LIN {X 0,Y 291.318,Z 1128.416,A -85,B 0,C 180,E1 14289.507,E2 14289.507} C_VEL
LIN {X 0,Y 294.597,Z 1120.605,A -85,B 0,C 180,E1 14284.989,E2 14284.989} C_VEL
LIN {X 0,Y 299.216,Z 1110.98,A -85,B 0,C 180,E1 14280.578,E2 14280.578} C_VEL
LIN {X 0,Y 304.532,Z 1100.924,A -85,B 0,C 180,E1 14276.748,E2 14276.748} C_VEL
LIN {X 0,Y 312.055,Z 1087.317,A -85,B 0,C 180,E1 14272.497,E2 14272.497} C_VEL
LIN {X 0,Y 318.965,Z 1075.015,A -85,B 0,C 180,E1 14269.304,E2 14269.304} C_VEL
LIN {X 0,Y 328.289,Z 1058.31,A -85,B 0,C 180,E1 14265.705,E2 14265.705} C_VEL
LIN {X 0,Y 336.427,Z 1043.264,A -85,B 0,C 180,E1 14263.018,E2 14263.018} C_VEL
LIN {X 0,Y 345.957,Z 1024.879,A -85,B 0,C 180,E1 14260.269,E2 14260.269} C_VEL
LIN {X 0,Y 354.466,Z 1007.296,A -85,B 0,C 180,E1 14258.092,E2 14258.092} C_VEL
LIN {X 0,Y 363.463,Z 987.421,A -85,B 0,C 180,E1 14256.021,E2 14256.021} C_VEL
LIN {X 0,Y 371.644,Z 967.379,A -85,B 0,C 180,E1 14254.313,E2 14254.313} C_VEL
LIN {X 0,Y 379.169,Z 947.195,A -85,B 0,C 180,E1 14252.87,E2 14252.87} C_VEL
LIN {X 0,Y 386.589,Z 924.342,A -85,B 0,C 180,E1 14251.544,E2 14251.544} C_VEL
LIN {X 0,Y 392.137,Z 904.806,A -85,B 0,C 180,E1 14250.618,E2 14250.618} C_VEL
LIN {X 0,Y 398.28,Z 879.112,A -85,B 0,C 180,E1 14249.658,E2 14249.658} C_VEL
LIN {X 0,Y 402.39,Z 857.399,A -85,B 0,C 180,E1 14249.039,E2 14249.039} C_VEL
LIN {X 0,Y 405.943,Z 831.436,A -85,B 0,C 180,E1 14248.465,E2 14248.465} C_VEL
LIN {X 0,Y 413.005,Z 740.206,A -85,B 0,C 180,E1 14246.94,E2 14246.94} C_VEL
LIN {X 0,Y 422.684,Z 613.309,A -85,B 0,C 180,E1 14244.865,E2 14244.865} C_VEL
LIN {X 0,Y 415.721,Z 599.338,A -85,B 0,C 180,E1 14242.298,E2 14242.298} C_VEL
LIN {X 0,Y 409.613,Z 587.739,A -85,B 0,C 180,E1 14239.76,E2 14239.76} C_VEL
LIN {X 0,Y 404.109,Z 578.023,A -85,B 0,C 180,E1 14237.161,E2 14237.161} C_VEL
LIN {X 0,Y 399.634,Z 571.534,A -85,B 0,C 180,E1 14234.786,E2 14234.786} C_VEL
LIN {X 0,Y 396.985,Z 567.648,A -85,B 0,C 180,E1 14233.176,E2 14233.176} C_VEL
LIN {X 0,Y 393.841,Z 563.029,A -85,B 0,C 180,E1 14230.977,E2 14230.977} C_VEL
LIN {X 0,Y 390.748,Z 558.424,A -85,B 0,C 180,E1 14228.313,E2 14228.313} C_VEL
LIN {X 0,Y 387.61,Z 554.339,A -85,B 0,C 180,E1 14224.587,E2 14224.587} C_VEL
LIN {X 0,Y 387.003,Z 552.755,A -85,B 0,C 180,E1 14223.407,E2 14223.407} C_VEL
LIN {X 0,Y 385.579,Z 551.937,A -85,B 0,C 180,E1 14217.325,E2 14217.325} C_VEL
LIN {X 0,Y 387.13,Z 552.997,A -85,B 0,C 180,E1 14212.804,E2 14212.804} C_VEL
LIN {X 0,Y 389.137,Z 556.879,A -85,B 0,C 180,E1 14209.778,E2 14209.778} C_VEL
LIN {X 0,Y 390.847,Z 558.677,A -85,B 0,C 180,E1 14208.04,E2 14208.04} C_VEL
LIN {X 0,Y 393.889,Z 563.127,A -85,B 0,C 180,E1 14205.445,E2 14205.445} C_VEL
LIN {X 0,Y 398.297,Z 569.544,A -85,B 0,C 180,E1 14202.467,E2 14202.467} C_VEL
LIN {X 0,Y 402.044,Z 575.153,A -85,B 0,C 180,E1 14200.344,E2 14200.344} C_VEL
LIN {X 0,Y 406.988,Z 582.534,A -85,B 0,C 180,E1 14197.92,E2 14197.92} C_VEL
LIN {X 0,Y 414.502,Z 594.463,A -85,B 0,C 180,E1 14194.752,E2 14194.752} C_VEL
LIN {X 0,Y 422.345,Z 607.879,A -85,B 0,C 180,E1 14191.892,E2 14191.892} C_VEL
LIN {X 0,Y 422.901,Z 609.086,A -85,B 0,C 180,E1 14191.695,E2 14191.695} C_VEL
LIN {X 0,Y 406.891,Z 815.861,A -85,B 0,C 180,E1 14188.311,E2 14188.311} C_VEL
LIN {X 0,Y 403.396,Z 842.508,A -85,B 0,C 180,E1 14187.705,E2 14187.705} C_VEL
LIN {X 0,Y 399.622,Z 863.558,A -85,B 0,C 180,E1 14187.058,E2 14187.058} C_VEL
LIN {X 0,Y 394.223,Z 887.589,A -85,B 0,C 180,E1 14186.117,E2 14186.117} C_VEL
LIN {X 0,Y 388.753,Z 907.638,A -85,B 0,C 180,E1 14185.134,E2 14185.134} C_VEL
LIN {X 0,Y 382.006,Z 929.3,A -85,B 0,C 180,E1 14183.852,E2 14183.852} C_VEL
LIN {X 0,Y 374.455,Z 950.085,A -85,B 0,C 180,E1 14182.348,E2 14182.348} C_VEL
LIN {X 0,Y 366.884,Z 968.981,A -85,B 0,C 180,E1 14180.715,E2 14180.715} C_VEL
LIN {X 0,Y 357.58,Z 989.896,A -85,B 0,C 180,E1 14178.539,E2 14178.539} C_VEL
LIN {X 0,Y 349.566,Z 1006.457,A -85,B 0,C 180,E1 14176.478,E2 14176.478} C_VEL
LIN {X 0,Y 339.978,Z 1024.981,A -85,B 0,C 180,E1 14173.721,E2 14173.721} C_VEL
LIN {X 0,Y 331.81,Z 1039.815,A -85,B 0,C 180,E1 14171.066,E2 14171.066} C_VEL
LIN {X 0,Y 323.054,Z 1055.197,A -85,B 0,C 180,E1 14167.795,E2 14167.795} C_VEL
LIN {X 0,Y 315.261,Z 1068.407,A -85,B 0,C 180,E1 14164.371,E2 14164.371} C_VEL
LIN {X 0,Y 307.881,Z 1081.062,A -85,B 0,C 180,E1 14160.44,E2 14160.44} C_VEL
LIN {X 0,Y 301.727,Z 1091.661,A -85,B 0,C 180,E1 14156.363,E2 14156.363} C_VEL
LIN {X 0,Y 296.66,Z 1101.087,A -85,B 0,C 180,E1 14151.97,E2 14151.97} C_VEL
LIN {X 0,Y 292.914,Z 1108.615,A -85,B 0,C 180,E1 14147.482,E2 14147.482} C_VEL
LIN {X 0,Y 290.432,Z 1114.59,A -85,B 0,C 180,E1 14143.016,E2 14143.016} C_VEL
LIN {X 0,Y 288.888,Z 1119.317,A -85,B 0,C 180,E1 14138.15,E2 14138.15} C_VEL
LIN {X 0,Y 288.298,Z 1121.988,A -85,B 0,C 180,E1 14134.177,E2 14134.177} C_VEL
LIN {X 0,Y 288.124,Z 1123.632,A -85,B 0,C 180,E1 14130.199,E2 14130.199} C_VEL
LIN {X 0,Y 288.073,Z 1124.223,A -85,B 0,C 180,E1 14125.621,E2 14125.621} C_VEL
LIN {X 0,Y 288.237,Z 1123.469,A -85,B 0,C 180,E1 14121.366,E2 14121.366} C_VEL
LIN {X 0,Y 288.657,Z 1121.74,A -85,B 0,C 180,E1 14117.395,E2 14117.395} C_VEL
LIN {X 0,Y 289.943,Z 1118.252,A -85,B 0,C 180,E1 14112.541,E2 14112.541} C_VEL
LIN {X 0,Y 292.111,Z 1113.467,A -85,B 0,C 180,E1 14108.069,E2 14108.069} C_VEL
LIN {X 0,Y 295.421,Z 1107.398,A -85,B 0,C 180,E1 14103.68,E2 14103.68} C_VEL
LIN {X 0,Y 300.504,Z 1098.901,A -85,B 0,C 180,E1 14098.953,E2 14098.953} C_VEL
LIN {X 0,Y 306.297,Z 1089.902,A -85,B 0,C 180,E1 14094.932,E2 14094.932} C_VEL
LIN {X 0,Y 314.024,Z 1078.102,A -85,B 0,C 180,E1 14090.681,E2 14090.681} C_VEL
LIN {X 0,Y 321.519,Z 1066.718,A -85,B 0,C 180,E1 14087.316,E2 14087.316} C_VEL
LIN {X 0,Y 331.369,Z 1051.399,A -85,B 0,C 180,E1 14083.598,E2 14083.598} C_VEL
LIN {X 0,Y 339.824,Z 1037.756,A -85,B 0,C 180,E1 14080.87,E2 14080.87} C_VEL
LIN {X 0,Y 350.085,Z 1020.363,A -85,B 0,C 180,E1 14077.973,E2 14077.973} C_VEL
LIN {X 0,Y 359.032,Z 1004.061,A -85,B 0,C 180,E1 14075.726,E2 14075.726} C_VEL
LIN {X 0,Y 368.488,Z 985.668,A -85,B 0,C 180,E1 14073.587,E2 14073.587} C_VEL
LIN {X 0,Y 377.392,Z 966.348,A -85,B 0,C 180,E1 14071.735,E2 14071.735} C_VEL
LIN {X 0,Y 385.777,Z 946.452,A -85,B 0,C 180,E1 14070.131,E2 14070.131} C_VEL
LIN {X 0,Y 393.826,Z 924.602,A -85,B 0,C 180,E1 14068.694,E2 14068.694} C_VEL
LIN {X 0,Y 400.441,Z 904.114,A -85,B 0,C 180,E1 14067.572,E2 14067.572} C_VEL
LIN {X 0,Y 407.002,Z 879.98,A -85,B 0,C 180,E1 14066.509,E2 14066.509} C_VEL
LIN {X 0,Y 411.754,Z 858.766,A -85,B 0,C 180,E1 14065.772,E2 14065.772} C_VEL
LIN {X 0,Y 416.215,Z 833.027,A -85,B 0,C 180,E1 14065.084,E2 14065.084} C_VEL
LIN {X 0,Y 417.621,Z 822.757,A -85,B 0,C 180,E1 14064.861,E2 14064.861} C_VEL
LIN {X 0,Y 418.116,Z 815.259,A -85,B 0,C 180,E1 14064.593,E2 14064.593} C_VEL
LIN {X 0,Y 417.112,Z 795.608,A -85,B 0,C 180,E1 14063.491,E2 14063.491} C_VEL
LIN {X 0,Y 417.306,Z 789.105,A -85,B 0,C 180,E1 14063.295,E2 14063.295} C_VEL
LIN {X 0,Y 431.206,Z 621.77,A -85,B 0,C 180,E1 14060.638,E2 14060.638} C_VEL
LIN {X 0,Y 425.225,Z 611.601,A -85,B 0,C 180,E1 14058.047,E2 14058.047} C_VEL
LIN {X 0,Y 420.08,Z 603.181,A -85,B 0,C 180,E1 14055.461,E2 14055.461} C_VEL
LIN {X 0,Y 415.509,Z 595.786,A -85,B 0,C 180,E1 14052.72,E2 14052.72} C_VEL
LIN {X 0,Y 412.212,Z 590.841,A -85,B 0,C 180,E1 14050.341,E2 14050.341} C_VEL
LIN {X 0,Y 409.345,Z 586.345,A -85,B 0,C 180,E1 14047.721,E2 14047.721} C_VEL
LIN {X 0,Y 406.77,Z 582.311,A -85,B 0,C 180,E1 14044.37,E2 14044.37} C_VEL
LIN {X 0,Y 406.343,Z 581.334,A -85,B 0,C 180,E1 14043.527,E2 14043.527} C_VEL
LIN {X 0,Y 405.047,Z 580.42,A -85,B 0,C 180,E1 14038.161,E2 14038.161} C_VEL
LIN {X 0,Y 406.537,Z 581.568,A -85,B 0,C 180,E1 14033.575,E2 14033.575} C_VEL
LIN {X 0,Y 408.82,Z 585.774,A -85,B 0,C 180,E1 14030.284,E2 14030.284} C_VEL
LIN {X 0,Y 409.908,Z 587.173,A -85,B 0,C 180,E1 14029.174,E2 14029.174} C_VEL
LIN {X 0,Y 413.207,Z 592.327,A -85,B 0,C 180,E1 14026.353,E2 14026.353} C_VEL
LIN {X 0,Y 416.68,Z 597.764,A -85,B 0,C 180,E1 14023.981,E2 14023.981} C_VEL
LIN {X 0,Y 421.249,Z 606.254,A -85,B 0,C 180,E1 14021.31,E2 14021.31} C_VEL
LIN {X 0,Y 426.021,Z 615.589,A -85,B 0,C 180,E1 14018.919,E2 14018.919} C_VEL
LIN {X 0,Y 431.055,Z 625.938,A -85,B 0,C 180,E1 14016.694,E2 14016.694} C_VEL
LIN {X 0,Y 414.036,Z 829.301,A -85,B 0,C 180,E1 14013.439,E2 14013.439} C_VEL
LIN {X 0,Y 410.198,Z 856.084,A -85,B 0,C 180,E1 14012.885,E2 14012.885} C_VEL
LIN {X 0,Y 405.917,Z 877.423,A -85,B 0,C 180,E1 14012.32,E2 14012.32} C_VEL
LIN {X 0,Y 399.909,Z 901.403,A -85,B 0,C 180,E1 14011.505,E2 14011.505} C_VEL
LIN {X 0,Y 393.63,Z 922.113,A -85,B 0,C 180,E1 14010.608,E2 14010.608} C_VEL
LIN {X 0,Y 386.08,Z 944.003,A -85,B 0,C 180,E1 14009.444,E2 14009.444} C_VEL
LIN {X 0,Y 377.335,Z 965.835,A -85,B 0,C 180,E1 14007.991,E2 14007.991} C_VEL
LIN {X 0,Y 368.463,Z 985.839,A -85,B 0,C 180,E1 14006.386,E2 14006.386} C_VEL
LIN {X 0,Y 358.485,Z 1006.049,A -85,B 0,C 180,E1 14004.396,E2 14004.396} C_VEL
LIN {X 0,Y 349.213,Z 1023.426,A -85,B 0,C 180,E1 14002.345,E2 14002.345} C_VEL
LIN {X 0,Y 338.447,Z 1042.153,A -85,B 0,C 180,E1 13999.661,E2 13999.661} C_VEL
LIN {X 0,Y 329.258,Z 1057.274,A -85,B 0,C 180,E1 13997.044,E2 13997.044} C_VEL
LIN {X 0,Y 318.775,Z 1073.827,A -85,B 0,C 180,E1 13993.567,E2 13993.567} C_VEL
LIN {X 0,Y 310.538,Z 1086.484,A -85,B 0,C 180,E1 13990.331,E2 13990.331} C_VEL
LIN {X 0,Y 301.758,Z 1099.978,A -85,B 0,C 180,E1 13986.144,E2 13986.144} C_VEL
LIN {X 0,Y 295.089,Z 1110.433,A -85,B 0,C 180,E1 13982.14,E2 13982.14} C_VEL
LIN {X 0,Y 289.07,Z 1120.545,A -85,B 0,C 180,E1 13977.39,E2 13977.39} C_VEL
LIN {X 0,Y 285.018,Z 1128.059,A -85,B 0,C 180,E1 13972.918,E2 13972.918} C_VEL
LIN {X 0,Y 282.106,Z 1134.694,A -85,B 0,C 180,E1 13967.961,E2 13967.961} C_VEL
LIN {X 0,Y 280.589,Z 1139.286,A -85,B 0,C 180,E1 13963.183,E2 13963.183} C_VEL
LIN {X 0,Y 280.078,Z 1142.124,A -85,B 0,C 180,E1 13959.038,E2 13959.038} C_VEL
LIN {X 0,Y 280.013,Z 1144.004,A -85,B 0,C 180,E1 13954.506,E2 13954.506} C_VEL
LIN {X 0,Y 280.074,Z 1144.409,A -85,B 0,C 180,E1 13950.205,E2 13950.205} C_VEL
LIN {X 0,Y 280.045,Z 1143.704,A -85,B 0,C 180,E1 13946.315,E2 13946.315} C_VEL
LIN {X 0,Y 280.021,Z 1142.095,A -85,B 0,C 180,E1 13942.614,E2 13942.614} C_VEL
LIN {X 0,Y 280.283,Z 1139.39,A -85,B 0,C 180,E1 13938.685,E2 13938.685} C_VEL
LIN {X 0,Y 281.319,Z 1134.776,A -85,B 0,C 180,E1 13933.905,E2 13933.905} C_VEL
LIN {X 0,Y 283.489,Z 1128.378,A -85,B 0,C 180,E1 13929.131,E2 13929.131} C_VEL
LIN {X 0,Y 286.643,Z 1121.177,A -85,B 0,C 180,E1 13924.813,E2 13924.813} C_VEL
LIN {X 0,Y 291.754,Z 1111.066,A -85,B 0,C 180,E1 13919.976,E2 13919.976} C_VEL
LIN {X 0,Y 297.297,Z 1101.056,A -85,B 0,C 180,E1 13916.061,E2 13916.061} C_VEL
LIN {X 0,Y 305.115,Z 1087.545,A -85,B 0,C 180,E1 13911.73,E2 13911.73} C_VEL
LIN {X 0,Y 312.276,Z 1075.296,A -85,B 0,C 180,E1 13908.486,E2 13908.486} C_VEL
LIN {X 0,Y 321.302,Z 1059.818,A -85,B 0,C 180,E1 13905.055,E2 13905.055} C_VEL
LIN {X 0,Y 329.779,Z 1044.674,A -85,B 0,C 180,E1 13902.285,E2 13902.285} C_VEL
LIN {X 0,Y 338.983,Z 1027.674,A -85,B 0,C 180,E1 13899.658,E2 13899.658} C_VEL
LIN {X 0,Y 348.447,Z 1008.81,A -85,B 0,C 180,E1 13897.263,E2 13897.263} C_VEL
LIN {X 0,Y 356.802,Z 991.001,A -85,B 0,C 180,E1 13895.364,E2 13895.364} C_VEL
LIN {X 0,Y 366.103,Z 969.234,A -85,B 0,C 180,E1 13893.449,E2 13893.449} C_VEL
LIN {X 0,Y 373.437,Z 950.196,A -85,B 0,C 180,E1 13892.065,E2 13892.065} C_VEL
LIN {X 0,Y 381.343,Z 927.037,A -85,B 0,C 180,E1 13890.68,E2 13890.68} C_VEL
LIN {X 0,Y 387.34,Z 906.608,A -85,B 0,C 180,E1 13889.697,E2 13889.697} C_VEL
LIN {X 0,Y 393.371,Z 882.74,A -85,B 0,C 180,E1 13888.777,E2 13888.777} C_VEL
LIN {X 0,Y 398.041,Z 859.048,A -85,B 0,C 180,E1 13888.091,E2 13888.091} C_VEL
LIN {X 0,Y 401.696,Z 834.331,A -85,B 0,C 180,E1 13887.53,E2 13887.53} C_VEL
LIN {X 0,Y 405.94,Z 782.941,A -85,B 0,C 180,E1 13886.658,E2 13886.658} C_VEL
LIN {X 0,Y 418.812,Z 617.464,A -85,B 0,C 180,E1 13883.945,E2 13883.945} C_VEL
LIN {X 0,Y 412.599,Z 604.766,A -85,B 0,C 180,E1 13881.54,E2 13881.54} C_VEL
LIN {X 0,Y 406.933,Z 593.772,A -85,B 0,C 180,E1 13879.075,E2 13879.075} C_VEL
LIN {X 0,Y 401.952,Z 584.841,A -85,B 0,C 180,E1 13876.623,E2 13876.623} C_VEL
LIN {X 0,Y 396.118,Z 575.974,A -85,B 0,C 180,E1 13873.28,E2 13873.28} C_VEL
LIN {X 0,Y 392.286,Z 570.526,A -85,B 0,C 180,E1 13870.575,E2 13870.575} C_VEL
LIN {X 0,Y 389.241,Z 565.913,A -85,B 0,C 180,E1 13867.825,E2 13867.825} C_VEL
LIN {X 0,Y 386.492,Z 562.133,A -85,B 0,C 180,E1 13864.377,E2 13864.377} C_VEL
LIN {X 0,Y 385.863,Z 560.619,A -85,B 0,C 180,E1 13863.119,E2 13863.119} C_VEL
LIN {X 0,Y 384.612,Z 559.887,A -85,B 0,C 180,E1 13857.238,E2 13857.238} C_VEL
LIN {X 0,Y 386.069,Z 560.932,A -85,B 0,C 180,E1 13852.933,E2 13852.933} C_VEL
LIN {X 0,Y 388.03,Z 564.753,A -85,B 0,C 180,E1 13849.908,E2 13849.908} C_VEL
LIN {X 0,Y 389.641,Z 566.527,A -85,B 0,C 180,E1 13848.228,E2 13848.228} C_VEL
LIN {X 0,Y 393.378,Z 572.138,A -85,B 0,C 180,E1 13845.049,E2 13845.049} C_VEL
LIN {X 0,Y 396.85,Z 577.291,A -85,B 0,C 180,E1 13842.704,E2 13842.704} C_VEL
LIN {X 0,Y 400.86,Z 583.4,A -85,B 0,C 180,E1 13840.397,E2 13840.397} C_VEL
LIN {X 0,Y 406.295,Z 591.861,A -85,B 0,C 180,E1 13837.72,E2 13837.72} C_VEL
LIN {X 0,Y 412.545,Z 602.045,A -85,B 0,C 180,E1 13835.056,E2 13835.056} C_VEL
LIN {X 0,Y 419.042,Z 613.451,A -85,B 0,C 180,E1 13832.606,E2 13832.606} C_VEL
LIN {X 0,Y 402.939,Z 816.204,A -85,B 0,C 180,E1 13829.295,E2 13829.295} C_VEL
LIN {X 0,Y 399.39,Z 842.701,A -85,B 0,C 180,E1 13828.695,E2 13828.695} C_VEL
LIN {X 0,Y 395.555,Z 863.662,A -85,B 0,C 180,E1 13828.055,E2 13828.055} C_VEL
LIN {X 0,Y 389.975,Z 887.969,A -85,B 0,C 180,E1 13827.109,E2 13827.109} C_VEL
LIN {X 0,Y 384.256,Z 908.433,A -85,B 0,C 180,E1 13826.108,E2 13826.108} C_VEL
LIN {X 0,Y 377.03,Z 930.975,A -85,B 0,C 180,E1 13824.768,E2 13824.768} C_VEL
LIN {X 0,Y 369.105,Z 952.049,A -85,B 0,C 180,E1 13823.224,E2 13823.224} C_VEL
LIN {X 0,Y 360.657,Z 972.488,A -85,B 0,C 180,E1 13821.428,E2 13821.428} C_VEL
LIN {X 0,Y 351.729,Z 991.656,A -85,B 0,C 180,E1 13819.379,E2 13819.379} C_VEL
LIN {X 0,Y 342.976,Z 1009.179,A -85,B 0,C 180,E1 13817.156,E2 13817.156} C_VEL
LIN {X 0,Y 333.519,Z 1026.666,A -85,B 0,C 180,E1 13814.477,E2 13814.477} C_VEL
LIN {X 0,Y 325.281,Z 1041.127,A -85,B 0,C 180,E1 13811.839,E2 13811.839} C_VEL
LIN {X 0,Y 315.828,Z 1057.018,A -85,B 0,C 180,E1 13808.355,E2 13808.355} C_VEL
LIN {X 0,Y 308.222,Z 1069.464,A -85,B 0,C 180,E1 13805.044,E2 13805.044} C_VEL
LIN {X 0,Y 300.268,Z 1082.475,A -85,B 0,C 180,E1 13800.852,E2 13800.852} C_VEL
LIN {X 0,Y 294.476,Z 1092.057,A -85,B 0,C 180,E1 13797.065,E2 13797.065} C_VEL
LIN {X 0,Y 289.158,Z 1101.46,A -85,B 0,C 180,E1 13792.571,E2 13792.571} C_VEL
LIN {X 0,Y 285.212,Z 1108.974,A -85,B 0,C 180,E1 13787.969,E2 13787.969} C_VEL
LIN {X 0,Y 282.551,Z 1115.04,A -85,B 0,C 180,E1 13783.298,E2 13783.298} C_VEL
LIN {X 0,Y 280.943,Z 1119.634,A -85,B 0,C 180,E1 13778.391,E2 13778.391} C_VEL
LIN {X 0,Y 280.316,Z 1122.299,A -85,B 0,C 180,E1 13774.296,E2 13774.296} C_VEL
LIN {X 0,Y 280.12,Z 1124,A -85,B 0,C 180,E1 13770,E2 13770} C_VEL
LIN {X 0,Y 280.077,Z 1124.503,A -85,B 0,C 180,E1 13765.495,E2 13765.495} C_VEL
LIN {X 0,Y 280.254,Z 1123.758,A -85,B 0,C 180,E1 13761.175,E2 13761.175} C_VEL
LIN {X 0,Y 280.723,Z 1122.003,A -85,B 0,C 180,E1 13757.033,E2 13757.033} C_VEL
LIN {X 0,Y 282.127,Z 1118.494,A -85,B 0,C 180,E1 13752.041,E2 13752.041} C_VEL
LIN {X 0,Y 284.457,Z 1113.728,A -85,B 0,C 180,E1 13747.471,E2 13747.471} C_VEL
LIN {X 0,Y 288.014,Z 1107.62,A -85,B 0,C 180,E1 13742.949,E2 13742.949} C_VEL
LIN {X 0,Y 293.416,Z 1099.099,A -85,B 0,C 180,E1 13738.116,E2 13738.116} C_VEL
LIN {X 0,Y 299.516,Z 1090.088,A -85,B 0,C 180,E1 13734.016,E2 13734.016} C_VEL
LIN {X 0,Y 307.628,Z 1078.261,A -85,B 0,C 180,E1 13729.698,E2 13729.698} C_VEL
LIN {X 0,Y 315.517,Z 1066.771,A -85,B 0,C 180,E1 13726.265,E2 13726.265} C_VEL
LIN {X 0,Y 325.7,Z 1051.512,A -85,B 0,C 180,E1 13722.541,E2 13722.541} C_VEL
LIN {X 0,Y 334.627,Z 1037.599,A -85,B 0,C 180,E1 13719.751,E2 13719.751} C_VEL
LIN {X 0,Y 345.645,Z 1019.407,A -85,B 0,C 180,E1 13716.744,E2 13716.744} C_VEL
LIN {X 0,Y 354.289,Z 1004.095,A -85,B 0,C 180,E1 13714.645,E2 13714.645} C_VEL
LIN {X 0,Y 364.331,Z 984.981,A -85,B 0,C 180,E1 13712.443,E2 13712.443} C_VEL
LIN {X 0,Y 373.15,Z 966.298,A -85,B 0,C 180,E1 13710.666,E2 13710.666} C_VEL
LIN {X 0,Y 381.967,Z 945.852,A -85,B 0,C 180,E1 13709.034,E2 13709.034} C_VEL
LIN {X 0,Y 389.918,Z 924.616,A -85,B 0,C 180,E1 13707.655,E2 13707.655} C_VEL
LIN {X 0,Y 396.746,Z 903.886,A -85,B 0,C 180,E1 13706.532,E2 13706.532} C_VEL
LIN {X 0,Y 403.264,Z 880.337,A -85,B 0,C 180,E1 13705.506,E2 13705.506} C_VEL
LIN {X 0,Y 408.135,Z 859.024,A -85,B 0,C 180,E1 13704.772,E2 13704.772} C_VEL
LIN {X 0,Y 412.708,Z 833.11,A -85,B 0,C 180,E1 13704.087,E2 13704.087} C_VEL
LIN {X 0,Y 415.407,Z 810.984,A -85,B 0,C 180,E1 13703.654,E2 13703.654} C_VEL
LIN {X 0,Y 417.306,Z 789.105,A -85,B 0,C 180,E1 13703.295,E2 13703.295} C_VEL
LIN {X 0,Y 417.512,Z 781.549,A -85,B 0,C 180,E1 13703.05,E2 13703.05} C_VEL
LIN {X 0,Y 416.613,Z 761.884,A -85,B 0,C 180,E1 13701.951,E2 13701.951} C_VEL
LIN {X 0,Y 416.864,Z 755.387,A -85,B 0,C 180,E1 13701.753,E2 13701.753} C_VEL
LIN {X 0,Y 427.803,Z 626.61,A -85,B 0,C 180,E1 13699.704,E2 13699.704} C_VEL
LIN {X 0,Y 421.397,Z 615.499,A -85,B 0,C 180,E1 13696.721,E2 13696.721} C_VEL
LIN {X 0,Y 416.189,Z 606.964,A -85,B 0,C 180,E1 13693.83,E2 13693.83} C_VEL
LIN {X 0,Y 413.107,Z 602.1,A -85,B 0,C 180,E1 13691.802,E2 13691.802} C_VEL
LIN {X 0,Y 410.882,Z 598.535,A -85,B 0,C 180,E1 13690.091,E2 13690.091} C_VEL
LIN {X 0,Y 408.093,Z 594.095,A -85,B 0,C 180,E1 13687.461,E2 13687.461} C_VEL
LIN {X 0,Y 405.602,Z 589.9,A -85,B 0,C 180,E1 13684.029,E2 13684.029} C_VEL
LIN {X 0,Y 405.215,Z 589.2,A -85,B 0,C 180,E1 13683.254,E2 13683.254} C_VEL
LIN {X 0,Y 404.072,Z 588.361,A -85,B 0,C 180,E1 13678.157,E2 13678.157} C_VEL
LIN {X 0,Y 405.481,Z 589.489,A -85,B 0,C 180,E1 13673.7,E2 13673.7} C_VEL
LIN {X 0,Y 407.849,Z 593.795,A -85,B 0,C 180,E1 13670.261,E2 13670.261} C_VEL
LIN {X 0,Y 408.78,Z 595.147,A -85,B 0,C 180,E1 13669.286,E2 13669.286} C_VEL
LIN {X 0,Y 411.86,Z 600.037,A -85,B 0,C 180,E1 13666.594,E2 13666.594} C_VEL
LIN {X 0,Y 415.156,Z 605.315,A -85,B 0,C 180,E1 13664.279,E2 13664.279} C_VEL
LIN {X 0,Y 419.675,Z 614.012,A -85,B 0,C 180,E1 13661.562,E2 13661.562} C_VEL
LIN {X 0,Y 424.084,Z 622.914,A -85,B 0,C 180,E1 13659.288,E2 13659.288} C_VEL
LIN {X 0,Y 427.699,Z 630.623,A -85,B 0,C 180,E1 13657.612,E2 13657.612} C_VEL
LIN {X 0,Y 410.688,Z 828.978,A -85,B 0,C 180,E1 13654.455,E2 13654.455} C_VEL
LIN {X 0,Y 406.787,Z 855.739,A -85,B 0,C 180,E1 13653.907,E2 13653.907} C_VEL
LIN {X 0,Y 402.42,Z 877.127,A -85,B 0,C 180,E1 13653.348,E2 13653.348} C_VEL
LIN {X 0,Y 396.146,Z 901.625,A -85,B 0,C 180,E1 13652.524,E2 13652.524} C_VEL
LIN {X 0,Y 389.747,Z 922.274,A -85,B 0,C 180,E1 13651.638,E2 13651.638} C_VEL
LIN {X 0,Y 381.681,Z 945.036,A -85,B 0,C 180,E1 13650.429,E2 13650.429} C_VEL
LIN {X 0,Y 372.956,Z 966.221,A -85,B 0,C 180,E1 13649.019,E2 13649.019} C_VEL
LIN {X 0,Y 363.433,Z 987.13,A -85,B 0,C 180,E1 13647.339,E2 13647.339} C_VEL
LIN {X 0,Y 353.473,Z 1006.609,A -85,B 0,C 180,E1 13645.404,E2 13645.404} C_VEL
LIN {X 0,Y 343.352,Z 1025.024,A -85,B 0,C 180,E1 13643.211,E2 13643.211} C_VEL
LIN {X 0,Y 332.609,Z 1042.975,A -85,B 0,C 180,E1 13640.588,E2 13640.588} C_VEL
LIN {X 0,Y 323.162,Z 1057.999,A -85,B 0,C 180,E1 13637.952,E2 13637.952} C_VEL
LIN {X 0,Y 312.409,Z 1074.294,A -85,B 0,C 180,E1 13634.461,E2 13634.461} C_VEL
LIN {X 0,Y 303.842,Z 1086.956,A -85,B 0,C 180,E1 13631.16,E2 13631.16} C_VEL
LIN {X 0,Y 294.734,Z 1100.306,A -85,B 0,C 180,E1 13626.904,E2 13626.904} C_VEL
LIN {X 0,Y 288.105,Z 1110.228,A -85,B 0,C 180,E1 13623.017,E2 13623.017} C_VEL
LIN {X 0,Y 281.748,Z 1120.319,A -85,B 0,C 180,E1 13618.165,E2 13618.165} C_VEL
LIN {X 0,Y 277.43,Z 1127.824,A -85,B 0,C 180,E1 13613.582,E2 13613.582} C_VEL
LIN {X 0,Y 274.313,Z 1134.442,A -85,B 0,C 180,E1 13608.489,E2 13608.489} C_VEL
LIN {X 0,Y 272.666,Z 1139.027,A -85,B 0,C 180,E1 13603.574,E2 13603.574} C_VEL
LIN {X 0,Y 272.091,Z 1141.858,A -85,B 0,C 180,E1 13599.305,E2 13599.305} C_VEL
LIN {X 0,Y 272.012,Z 1143.731,A -85,B 0,C 180,E1 13594.639,E2 13594.639} C_VEL
LIN {X 0,Y 272.079,Z 1144.12,A -85,B 0,C 180,E1 13590.211,E2 13590.211} C_VEL
LIN {X 0,Y 272.049,Z 1143.407,A -85,B 0,C 180,E1 13586.207,E2 13586.207} C_VEL
LIN {X 0,Y 272.025,Z 1141.787,A -85,B 0,C 180,E1 13582.396,E2 13582.396} C_VEL
LIN {X 0,Y 272.322,Z 1139.071,A -85,B 0,C 180,E1 13578.349,E2 13578.349} C_VEL
LIN {X 0,Y 273.507,Z 1134.284,A -85,B 0,C 180,E1 13573.301,E2 13573.301} C_VEL
LIN {X 0,Y 275.802,Z 1128.026,A -85,B 0,C 180,E1 13568.521,E2 13568.521} C_VEL
LIN {X 0,Y 279.356,Z 1120.449,A -85,B 0,C 180,E1 13563.88,E2 13563.88} C_VEL
LIN {X 0,Y 284.586,Z 1110.681,A -85,B 0,C 180,E1 13559.138,E2 13559.138} C_VEL
LIN {X 0,Y 290.43,Z 1100.658,A -85,B 0,C 180,E1 13555.145,E2 13555.145} C_VEL
LIN {X 0,Y 298.621,Z 1087.123,A -85,B 0,C 180,E1 13550.74,E2 13550.74} C_VEL
LIN {X 0,Y 306.096,Z 1074.862,A -85,B 0,C 180,E1 13547.454,E2 13547.454} C_VEL
LIN {X 0,Y 315.677,Z 1059.008,A -85,B 0,C 180,E1 13543.922,E2 13543.922} C_VEL
LIN {X 0,Y 324.261,Z 1044.194,A -85,B 0,C 180,E1 13541.201,E2 13541.201} C_VEL
LIN {X 0,Y 333.927,Z 1026.89,A -85,B 0,C 180,E1 13538.523,E2 13538.523} C_VEL
LIN {X 0,Y 343.609,Z 1008.08,A -85,B 0,C 180,E1 13536.146,E2 13536.146} C_VEL
LIN {X 0,Y 352.747,Z 989.085,A -85,B 0,C 180,E1 13534.137,E2 13534.137} C_VEL
LIN {X 0,Y 361.984,Z 967.796,A -85,B 0,C 180,E1 13532.301,E2 13532.301} C_VEL
LIN {X 0,Y 369.508,Z 948.636,A -85,B 0,C 180,E1 13530.929,E2 13530.929} C_VEL
LIN {X 0,Y 377.607,Z 925.152,A -85,B 0,C 180,E1 13529.557,E2 13529.557} C_VEL
LIN {X 0,Y 383.385,Z 905.806,A -85,B 0,C 180,E1 13528.644,E2 13528.644} C_VEL
LIN {X 0,Y 389.481,Z 882.018,A -85,B 0,C 180,E1 13527.741,E2 13527.741} C_VEL
LIN {X 0,Y 394.176,Z 858.584,A -85,B 0,C 180,E1 13527.07,E2 13527.07} C_VEL
LIN {X 0,Y 397.887,Z 833.863,A -85,B 0,C 180,E1 13526.514,E2 13526.514} C_VEL
LIN {X 0,Y 402.316,Z 781.445,A -85,B 0,C 180,E1 13525.628,E2 13525.628} C_VEL
LIN {X 0,Y 415.089,Z 621.78,A -85,B 0,C 180,E1 13523.027,E2 13523.027} C_VEL
LIN {X 0,Y 409.386,Z 609.849,A -85,B 0,C 180,E1 13520.699,E2 13520.699} C_VEL
LIN {X 0,Y 404.231,Z 599.763,A -85,B 0,C 180,E1 13518.346,E2 13518.346} C_VEL
LIN {X 0,Y 400.018,Z 592.019,A -85,B 0,C 180,E1 13516.183,E2 13516.183} C_VEL
LIN {X 0,Y 394.574,Z 583.529,A -85,B 0,C 180,E1 13512.96,E2 13512.96} C_VEL
LIN {X 0,Y 390.844,Z 578.114,A -85,B 0,C 180,E1 13510.242,E2 13510.242} C_VEL
LIN {X 0,Y 387.969,Z 573.664,A -85,B 0,C 180,E1 13507.553,E2 13507.553} C_VEL
LIN {X 0,Y 385.303,Z 569.721,A -85,B 0,C 180,E1 13504.018,E2 13504.018} C_VEL
LIN {X 0,Y 384.809,Z 568.525,A -85,B 0,C 180,E1 13502.979,E2 13502.979} C_VEL
LIN {X 0,Y 383.645,Z 567.837,A -85,B 0,C 180,E1 13497.162,E2 13497.162} C_VEL
LIN {X 0,Y 385.011,Z 568.863,A -85,B 0,C 180,E1 13493.064,E2 13493.064} C_VEL
LIN {X 0,Y 387.059,Z 572.778,A -85,B 0,C 180,E1 13489.883,E2 13489.883} C_VEL
LIN {X 0,Y 388.44,Z 574.374,A -85,B 0,C 180,E1 13488.417,E2 13488.417} C_VEL
LIN {X 0,Y 392.011,Z 579.857,A -85,B 0,C 180,E1 13485.298,E2 13485.298} C_VEL
LIN {X 0,Y 395.411,Z 585.033,A -85,B 0,C 180,E1 13482.942,E2 13482.942} C_VEL
LIN {X 0,Y 400.208,Z 592.352,A -85,B 0,C 180,E1 13480.174,E2 13480.174} C_VEL
LIN {X 0,Y 406.317,Z 602.391,A -85,B 0,C 180,E1 13477.195,E2 13477.195} C_VEL
LIN {X 0,Y 412.267,Z 612.537,A -85,B 0,C 180,E1 13474.693,E2 13474.693} C_VEL
LIN {X 0,Y 415.262,Z 618.162,A -85,B 0,C 180,E1 13473.528,E2 13473.528} C_VEL
LIN {X 0,Y 399.107,Z 816.538,A -85,B 0,C 180,E1 13470.297,E2 13470.297} C_VEL
LIN {X 0,Y 395.484,Z 843.014,A -85,B 0,C 180,E1 13469.702,E2 13469.702} C_VEL
LIN {X 0,Y 391.589,Z 863.864,A -85,B 0,C 180,E1 13469.07,E2 13469.07} C_VEL
LIN {X 0,Y 386.063,Z 887.562,A -85,B 0,C 180,E1 13468.159,E2 13468.159} C_VEL
LIN {X 0,Y 380.21,Z 908.113,A -85,B 0,C 180,E1 13467.165,E2 13467.165} C_VEL
LIN {X 0,Y 373.146,Z 929.789,A -85,B 0,C 180,E1 13465.895,E2 13465.895} C_VEL
LIN {X 0,Y 364.901,Z 951.391,A -85,B 0,C 180,E1 13464.337,E2 13464.337} C_VEL
LIN {X 0,Y 356.951,Z 970.219,A -85,B 0,C 180,E1 13462.707,E2 13462.707} C_VEL
LIN {X 0,Y 347.576,Z 990.162,A -85,B 0,C 180,E1 13460.628,E2 13460.628} C_VEL
LIN {X 0,Y 338.958,Z 1006.994,A -85,B 0,C 180,E1 13458.528,E2 13458.528} C_VEL
LIN {X 0,Y 328.493,Z 1025.983,A -85,B 0,C 180,E1 13455.669,E2 13455.669} C_VEL
LIN {X 0,Y 319.786,Z 1040.782,A -85,B 0,C 180,E1 13452.971,E2 13452.971} C_VEL
LIN {X 0,Y 310.411,Z 1056.098,A -85,B 0,C 180,E1 13449.628,E2 13449.628} C_VEL
LIN {X 0,Y 302.402,Z 1068.659,A -85,B 0,C 180,E1 13446.289,E2 13446.289} C_VEL
LIN {X 0,Y 294.674,Z 1080.842,A -85,B 0,C 180,E1 13442.421,E2 13442.421} C_VEL
LIN {X 0,Y 287.829,Z 1091.56,A -85,B 0,C 180,E1 13438.194,E2 13438.194} C_VEL
LIN {X 0,Y 282.561,Z 1100.291,A -85,B 0,C 180,E1 13434.013,E2 13434.013} C_VEL
LIN {X 0,Y 277.84,Z 1108.744,A -85,B 0,C 180,E1 13428.899,E2 13428.899} C_VEL
LIN {X 0,Y 275.12,Z 1114.399,A -85,B 0,C 180,E1 13424.523,E2 13424.523} C_VEL
LIN {X 0,Y 273.155,Z 1119.495,A -85,B 0,C 180,E1 13419.269,E2 13419.269} C_VEL
LIN {X 0,Y 272.383,Z 1122.39,A -85,B 0,C 180,E1 13414.843,E2 13414.843} C_VEL
LIN {X 0,Y 272.127,Z 1124.034,A -85,B 0,C 180,E1 13410.842,E2 13410.842} C_VEL
LIN {X 0,Y 272.075,Z 1124.772,A -85,B 0,C 180,E1 13406.629,E2 13406.629} C_VEL
LIN {X 0,Y 272.2,Z 1124.353,A -85,B 0,C 180,E1 13401.976,E2 13401.976} C_VEL
LIN {X 0,Y 272.654,Z 1122.7,A -85,B 0,C 180,E1 13397.504,E2 13397.504} C_VEL
LIN {X 0,Y 273.717,Z 1120.009,A -85,B 0,C 180,E1 13393.155,E2 13393.155} C_VEL
LIN {X 0,Y 276.175,Z 1115.2,A -85,B 0,C 180,E1 13387.881,E2 13387.881} C_VEL
LIN {X 0,Y 279.666,Z 1109.324,A -85,B 0,C 180,E1 13383.225,E2 13383.225} C_VEL
LIN {X 0,Y 284.801,Z 1101.69,A -85,B 0,C 180,E1 13378.458,E2 13378.458} C_VEL
LIN {X 0,Y 291.175,Z 1092.539,A -85,B 0,C 180,E1 13374.04,E2 13374.04} C_VEL
LIN {X 0,Y 298.579,Z 1082.3,A -85,B 0,C 180,E1 13369.986,E2 13369.986} C_VEL
LIN {X 0,Y 307.251,Z 1070.158,A -85,B 0,C 180,E1 13366.118,E2 13366.118} C_VEL
LIN {X 0,Y 315.854,Z 1057.916,A -85,B 0,C 180,E1 13362.892,E2 13362.892} C_VEL
LIN {X 0,Y 326.484,Z 1042.158,A -85,B 0,C 180,E1 13359.486,E2 13359.486} C_VEL
LIN {X 0,Y 335.456,Z 1028.118,A -85,B 0,C 180,E1 13356.981,E2 13356.981} C_VEL
LIN {X 0,Y 346.242,Z 1010.231,A -85,B 0,C 180,E1 13354.318,E2 13354.318} C_VEL
LIN {X 0,Y 356.05,Z 992.417,A -85,B 0,C 180,E1 13352.145,E2 13352.145} C_VEL
LIN {X 0,Y 365.991,Z 972.877,A -85,B 0,C 180,E1 13350.153,E2 13350.153} C_VEL
LIN {X 0,Y 374.897,Z 953.096,A -85,B 0,C 180,E1 13348.5,E2 13348.5} C_VEL
LIN {X 0,Y 383.402,Z 932.221,A -85,B 0,C 180,E1 13347.049,E2 13347.049} C_VEL
LIN {X 0,Y 390.986,Z 910.474,A -85,B 0,C 180,E1 13345.816,E2 13345.816} C_VEL
LIN {X 0,Y 396.881,Z 891.067,A -85,B 0,C 180,E1 13344.909,E2 13344.909} C_VEL
LIN {X 0,Y 403.105,Z 866.485,A -85,B 0,C 180,E1 13343.984,E2 13343.984} C_VEL
LIN {X 0,Y 407.318,Z 845.379,A -85,B 0,C 180,E1 13343.366,E2 13343.366} C_VEL
LIN {X 0,Y 411.06,Z 820.861,A -85,B 0,C 180,E1 13342.816,E2 13342.816} C_VEL
LIN {X 0,Y 415.87,Z 767.134,A -85,B 0,C 180,E1 13341.938,E2 13341.938} C_VEL
LIN {X 0,Y 416.864,Z 755.387,A -85,B 0,C 180,E1 13341.753,E2 13341.753} C_VEL
LIN {X 0,Y 417.112,Z 747.832,A -85,B 0,C 180,E1 13341.507,E2 13341.507} C_VEL
LIN {X 0,Y 416.409,Z 728.183,A -85,B 0,C 180,E1 13340.397,E2 13340.397} C_VEL
LIN {X 0,Y 416.7,Z 721.685,A -85,B 0,C 180,E1 13340.201,E2 13340.201} C_VEL
LIN {X 0,Y 424.554,Z 631.643,A -85,B 0,C 180,E1 13338.777,E2 13338.777} C_VEL
LIN {X 0,Y 418.914,Z 621.735,A -85,B 0,C 180,E1 13336.003,E2 13336.003} C_VEL
LIN {X 0,Y 414.212,Z 613.848,A -85,B 0,C 180,E1 13333.257,E2 13333.257} C_VEL
LIN {X 0,Y 411.453,Z 609.352,A -85,B 0,C 180,E1 13331.352,E2 13331.352} C_VEL
LIN {X 0,Y 409.476,Z 606.124,A -85,B 0,C 180,E1 13329.771,E2 13329.771} C_VEL
LIN {X 0,Y 406.982,Z 601.97,A -85,B 0,C 180,E1 13327.34,E2 13327.34} C_VEL
LIN {X 0,Y 404.51,Z 597.696,A -85,B 0,C 180,E1 13323.827,E2 13323.827} C_VEL
LIN {X 0,Y 404.097,Z 597.066,A -85,B 0,C 180,E1 13322.979,E2 13322.979} C_VEL
LIN {X 0,Y 403.106,Z 596.316,A -85,B 0,C 180,E1 13318.01,E2 13318.01} C_VEL
LIN {X 0,Y 404.427,Z 597.407,A -85,B 0,C 180,E1 13313.826,E2 13313.826} C_VEL
LIN {X 0,Y 406.747,Z 601.677,A -85,B 0,C 180,E1 13310.377,E2 13310.377} C_VEL
LIN {X 0,Y 407.654,Z 603.114,A -85,B 0,C 180,E1 13309.4,E2 13309.4} C_VEL
LIN {X 0,Y 410.52,Z 607.744,A -85,B 0,C 180,E1 13306.836,E2 13306.836} C_VEL
LIN {X 0,Y 413.643,Z 612.866,A -85,B 0,C 180,E1 13304.579,E2 13304.579} C_VEL
LIN {X 0,Y 418.347,Z 622.233,A -85,B 0,C 180,E1 13301.681,E2 13301.681} C_VEL
LIN {X 0,Y 423.857,Z 633.728,A -85,B 0,C 180,E1 13298.843,E2 13298.843} C_VEL
LIN {X 0,Y 424.445,Z 635.363,A -85,B 0,C 180,E1 13298.547,E2 13298.547} C_VEL
LIN {X 0,Y 407.454,Z 828.843,A -85,B 0,C 180,E1 13295.484,E2 13295.484} C_VEL
LIN {X 0,Y 403.488,Z 855.505,A -85,B 0,C 180,E1 13294.943,E2 13294.943} C_VEL
LIN {X 0,Y 399.043,Z 876.886,A -85,B 0,C 180,E1 13294.393,E2 13294.393} C_VEL
LIN {X 0,Y 392.511,Z 901.848,A -85,B 0,C 180,E1 13293.563,E2 13293.563} C_VEL
LIN {X 0,Y 385.993,Z 922.435,A -85,B 0,C 180,E1 13292.689,E2 13292.689} C_VEL
LIN {X 0,Y 377.765,Z 945.105,A -85,B 0,C 180,E1 13291.493,E2 13291.493} C_VEL
LIN {X 0,Y 369.012,Z 965.904,A -85,B 0,C 180,E1 13290.122,E2 13290.122} C_VEL
LIN {X 0,Y 359.463,Z 986.41,A -85,B 0,C 180,E1 13288.492,E2 13288.492} C_VEL
LIN {X 0,Y 349.141,Z 1006.138,A -85,B 0,C 180,E1 13286.552,E2 13286.552} C_VEL
LIN {X 0,Y 339.149,Z 1023.841,A -85,B 0,C 180,E1 13284.461,E2 13284.461} C_VEL
LIN {X 0,Y 328.05,Z 1041.936,A -85,B 0,C 180,E1 13281.849,E2 13281.849} C_VEL
LIN {X 0,Y 318.252,Z 1057.023,A -85,B 0,C 180,E1 13279.216,E2 13279.216} C_VEL
LIN {X 0,Y 307.141,Z 1073.319,A -85,B 0,C 180,E1 13275.742,E2 13275.742} C_VEL
LIN {X 0,Y 298.103,Z 1086.145,A -85,B 0,C 180,E1 13272.392,E2 13272.392} C_VEL
LIN {X 0,Y 288.526,Z 1099.59,A -85,B 0,C 180,E1 13268.088,E2 13268.088} C_VEL
LIN {X 0,Y 281.506,Z 1109.557,A -85,B 0,C 180,E1 13264.139,E2 13264.139} C_VEL
LIN {X 0,Y 274.963,Z 1119.371,A -85,B 0,C 180,E1 13259.401,E2 13259.401} C_VEL
LIN {X 0,Y 270.056,Z 1127.278,A -85,B 0,C 180,E1 13254.5,E2 13254.5} C_VEL
LIN {X 0,Y 266.754,Z 1133.699,A -85,B 0,C 180,E1 13249.488,E2 13249.488} C_VEL
LIN {X 0,Y 264.805,Z 1138.6,A -85,B 0,C 180,E1 13244.208,E2 13244.208} C_VEL
LIN {X 0,Y 264.126,Z 1141.472,A -85,B 0,C 180,E1 13239.808,E2 13239.808} C_VEL
LIN {X 0,Y 264.003,Z 1143.314,A -85,B 0,C 180,E1 13235.215,E2 13235.215} C_VEL
LIN {X 0,Y 264.074,Z 1143.875,A -85,B 0,C 180,E1 13230.651,E2 13230.651} C_VEL
LIN {X 0,Y 264.054,Z 1143.178,A -85,B 0,C 180,E1 13226.309,E2 13226.309} C_VEL
LIN {X 0,Y 264.028,Z 1141.596,A -85,B 0,C 180,E1 13222.383,E2 13222.383} C_VEL
LIN {X 0,Y 264.336,Z 1138.917,A -85,B 0,C 180,E1 13218.214,E2 13218.214} C_VEL
LIN {X 0,Y 265.54,Z 1134.338,A -85,B 0,C 180,E1 13213.145,E2 13213.145} C_VEL
LIN {X 0,Y 268.004,Z 1127.987,A -85,B 0,C 180,E1 13208.094,E2 13208.094} C_VEL
LIN {X 0,Y 271.616,Z 1120.663,A -85,B 0,C 180,E1 13203.451,E2 13203.451} C_VEL
LIN {X 0,Y 277.206,Z 1110.766,A -85,B 0,C 180,E1 13198.465,E2 13198.465} C_VEL
LIN {X 0,Y 283.302,Z 1100.789,A -85,B 0,C 180,E1 13194.384,E2 13194.384} C_VEL
LIN {X 0,Y 291.816,Z 1087.351,A -85,B 0,C 180,E1 13189.896,E2 13189.896} C_VEL
LIN {X 0,Y 299.563,Z 1075.143,A -85,B 0,C 180,E1 13186.56,E2 13186.56} C_VEL
LIN {X 0,Y 309.257,Z 1059.753,A -85,B 0,C 180,E1 13183.054,E2 13183.054} C_VEL
LIN {X 0,Y 318.86,Z 1043.714,A -85,B 0,C 180,E1 13180.08,E2 13180.08} C_VEL
LIN {X 0,Y 328.97,Z 1026.151,A -85,B 0,C 180,E1 13177.361,E2 13177.361} C_VEL
LIN {X 0,Y 338.83,Z 1007.503,A -85,B 0,C 180,E1 13175.015,E2 13175.015} C_VEL
LIN {X 0,Y 348.198,Z 988.526,A -85,B 0,C 180,E1 13173.016,E2 13173.016} C_VEL
LIN {X 0,Y 357.205,Z 968.298,A -85,B 0,C 180,E1 13171.278,E2 13171.278} C_VEL
LIN {X 0,Y 364.984,Z 948.986,A -85,B 0,C 180,E1 13169.896,E2 13169.896} C_VEL
LIN {X 0,Y 373.292,Z 925.553,A -85,B 0,C 180,E1 13168.529,E2 13168.529} C_VEL
LIN {X 0,Y 379.185,Z 906.301,A -85,B 0,C 180,E1 13167.623,E2 13167.623} C_VEL
LIN {X 0,Y 385.397,Z 882.768,A -85,B 0,C 180,E1 13166.729,E2 13166.729} C_VEL
LIN {X 0,Y 390.331,Z 858.723,A -85,B 0,C 180,E1 13166.044,E2 13166.044} C_VEL
LIN {X 0,Y 394.118,Z 834.2,A -85,B 0,C 180,E1 13165.494,E2 13165.494} C_VEL
LIN {X 0,Y 398.31,Z 786.317,A -85,B 0,C 180,E1 13164.684,E2 13164.684} C_VEL
LIN {X 0,Y 411.428,Z 626,A -85,B 0,C 180,E1 13162.075,E2 13162.075} C_VEL
LIN {X 0,Y 405.976,Z 614.451,A -85,B 0,C 180,E1 13159.72,E2 13159.72} C_VEL
LIN {X 0,Y 400.48,Z 603.441,A -85,B 0,C 180,E1 13157.022,E2 13157.022} C_VEL
LIN {X 0,Y 397.6,Z 598.453,A -85,B 0,C 180,E1 13155.46,E2 13155.46} C_VEL
LIN {X 0,Y 392.933,Z 590.954,A -85,B 0,C 180,E1 13152.566,E2 13152.566} C_VEL
LIN {X 0,Y 389.503,Z 585.803,A -85,B 0,C 180,E1 13149.979,E2 13149.979} C_VEL
LIN {X 0,Y 386.707,Z 581.415,A -85,B 0,C 180,E1 13147.279,E2 13147.279} C_VEL
LIN {X 0,Y 384.165,Z 577.411,A -85,B 0,C 180,E1 13143.731,E2 13143.731} C_VEL
LIN {X 0,Y 383.758,Z 576.432,A -85,B 0,C 180,E1 13142.838,E2 13142.838} C_VEL
LIN {X 0,Y 382.67,Z 575.779,A -85,B 0,C 180,E1 13137.154,E2 13137.154} C_VEL
LIN {X 0,Y 383.955,Z 576.791,A -85,B 0,C 180,E1 13133.195,E2 13133.195} C_VEL
LIN {X 0,Y 386.088,Z 580.8,A -85,B 0,C 180,E1 13129.857,E2 13129.857} C_VEL
LIN {X 0,Y 387.243,Z 582.218,A -85,B 0,C 180,E1 13128.607,E2 13128.607} C_VEL
LIN {X 0,Y 390.651,Z 587.572,A -85,B 0,C 180,E1 13125.549,E2 13125.549} C_VEL
LIN {X 0,Y 393.872,Z 592.591,A -85,B 0,C 180,E1 13123.254,E2 13123.254} C_VEL
LIN {X 0,Y 398.498,Z 599.852,A -85,B 0,C 180,E1 13120.505,E2 13120.505} C_VEL
LIN {X 0,Y 404.338,Z 609.671,A -85,B 0,C 180,E1 13117.577,E2 13117.577} C_VEL
LIN {X 0,Y 410.079,Z 619.723,A -85,B 0,C 180,E1 13115.091,E2 13115.091} C_VEL
LIN {X 0,Y 411.607,Z 622.679,A -85,B 0,C 180,E1 13114.47,E2 13114.47} C_VEL
LIN {X 0,Y 395.416,Z 816.709,A -85,B 0,C 180,E1 13111.322,E2 13111.322} C_VEL
LIN {X 0,Y 391.702,Z 843.327,A -85,B 0,C 180,E1 13110.727,E2 13110.727} C_VEL
LIN {X 0,Y 387.726,Z 864.173,A -85,B 0,C 180,E1 13110.101,E2 13110.101} C_VEL
LIN {X 0,Y 381.926,Z 888.42,A -85,B 0,C 180,E1 13109.173,E2 13109.173} C_VEL
LIN {X 0,Y 375.951,Z 908.903,A -85,B 0,C 180,E1 13108.185,E2 13108.185} C_VEL
LIN {X 0,Y 368.392,Z 931.468,A -85,B 0,C 180,E1 13106.86,E2 13106.86} C_VEL
LIN {X 0,Y 360.297,Z 952.042,A -85,B 0,C 180,E1 13105.371,E2 13105.371} C_VEL
LIN {X 0,Y 351.835,Z 971.561,A -85,B 0,C 180,E1 13103.677,E2 13103.677} C_VEL
LIN {X 0,Y 342.092,Z 991.586,A -85,B 0,C 180,E1 13101.567,E2 13101.567} C_VEL
LIN {X 0,Y 333.096,Z 1008.624,A -85,B 0,C 180,E1 13099.417,E2 13099.417} C_VEL
LIN {X 0,Y 322.901,Z 1026.482,A -85,B 0,C 180,E1 13096.694,E2 13096.694} C_VEL
LIN {X 0,Y 313.916,Z 1041.264,A -85,B 0,C 180,E1 13093.978,E2 13093.978} C_VEL
LIN {X 0,Y 303.752,Z 1057.234,A -85,B 0,C 180,E1 13090.428,E2 13090.428} C_VEL
LIN {X 0,Y 295.33,Z 1069.963,A -85,B 0,C 180,E1 13086.963,E2 13086.963} C_VEL
LIN {X 0,Y 286.798,Z 1082.79,A -85,B 0,C 180,E1 13082.71,E2 13082.71} C_VEL
LIN {X 0,Y 280.12,Z 1092.848,A -85,B 0,C 180,E1 13078.576,E2 13078.576} C_VEL
LIN {X 0,Y 274.26,Z 1102.202,A -85,B 0,C 180,E1 13073.871,E2 13073.871} C_VEL
LIN {X 0,Y 269.874,Z 1109.691,A -85,B 0,C 180,E1 13069.029,E2 13069.029} C_VEL
LIN {X 0,Y 266.818,Z 1115.92,A -85,B 0,C 180,E1 13063.928,E2 13063.928} C_VEL
LIN {X 0,Y 265.063,Z 1120.28,A -85,B 0,C 180,E1 13058.897,E2 13058.897} C_VEL
LIN {X 0,Y 264.355,Z 1122.922,A -85,B 0,C 180,E1 13054.556,E2 13054.556} C_VEL
LIN {X 0,Y 264.131,Z 1124.6,A -85,B 0,C 180,E1 13050,E2 13050} C_VEL
LIN {X 0,Y 264.088,Z 1125.063,A -85,B 0,C 180,E1 13045.222,E2 13045.222} C_VEL
LIN {X 0,Y 264.286,Z 1124.365,A -85,B 0,C 180,E1 13040.857,E2 13040.857} C_VEL
LIN {X 0,Y 264.798,Z 1122.745,A -85,B 0,C 180,E1 13036.683,E2 13036.683} C_VEL
LIN {X 0,Y 266.281,Z 1119.544,A -85,B 0,C 180,E1 13031.614,E2 13031.614} C_VEL
LIN {X 0,Y 269.125,Z 1114.442,A -85,B 0,C 180,E1 13026.343,E2 13026.343} C_VEL
LIN {X 0,Y 272.922,Z 1108.658,A -85,B 0,C 180,E1 13021.796,E2 13021.796} C_VEL
LIN {X 0,Y 279.03,Z 1100.066,A -85,B 0,C 180,E1 13016.611,E2 13016.611} C_VEL
LIN {X 0,Y 285.501,Z 1091.368,A -85,B 0,C 180,E1 13012.455,E2 13012.455} C_VEL
LIN {X 0,Y 294.709,Z 1079.149,A -85,B 0,C 180,E1 13007.795,E2 13007.795} C_VEL
LIN {X 0,Y 303.17,Z 1067.784,A -85,B 0,C 180,E1 13004.3,E2 13004.3} C_VEL
LIN {X 0,Y 314.194,Z 1052.504,A -85,B 0,C 180,E1 13000.482,E2 13000.482} C_VEL
LIN {X 0,Y 323.548,Z 1038.886,A -85,B 0,C 180,E1 12997.707,E2 12997.707} C_VEL
LIN {X 0,Y 334.803,Z 1021.545,A -85,B 0,C 180,E1 12994.786,E2 12994.786} C_VEL
LIN {X 0,Y 344.55,Z 1005.273,A -85,B 0,C 180,E1 12992.537,E2 12992.537} C_VEL
LIN {X 0,Y 354.785,Z 986.942,A -85,B 0,C 180,E1 12990.413,E2 12990.413} C_VEL
LIN {X 0,Y 364.374,Z 967.676,A -85,B 0,C 180,E1 12988.583,E2 12988.583} C_VEL
LIN {X 0,Y 372.869,Z 948.944,A -85,B 0,C 180,E1 12987.089,E2 12987.089} C_VEL
LIN {X 0,Y 381.596,Z 927.117,A -85,B 0,C 180,E1 12985.66,E2 12985.66} C_VEL
LIN {X 0,Y 388.63,Z 906.839,A -85,B 0,C 180,E1 12984.562,E2 12984.562} C_VEL
LIN {X 0,Y 395.792,Z 882.541,A -85,B 0,C 180,E1 12983.501,E2 12983.501} C_VEL
LIN {X 0,Y 400.974,Z 860.945,A -85,B 0,C 180,E1 12982.763,E2 12982.763} C_VEL
LIN {X 0,Y 405.571,Z 836.84,A -85,B 0,C 180,E1 12982.12,E2 12982.12} C_VEL
LIN {X 0,Y 408.647,Z 813.312,A -85,B 0,C 180,E1 12981.656,E2 12981.656} C_VEL
LIN {X 0,Y 416.7,Z 721.685,A -85,B 0,C 180,E1 12980.201,E2 12980.201} C_VEL
LIN {X 0,Y 416.999,Z 714.132,A -85,B 0,C 180,E1 12979.957,E2 12979.957} C_VEL
LIN {X 0,Y 416.506,Z 694.493,A -85,B 0,C 180,E1 12978.842,E2 12978.842} C_VEL
LIN {X 0,Y 416.828,Z 687.998,A -85,B 0,C 180,E1 12978.644,E2 12978.644} C_VEL
LIN {X 0,Y 421.387,Z 636.678,A -85,B 0,C 180,E1 12977.824,E2 12977.824} C_VEL
LIN {X 0,Y 415.75,Z 626.529,A -85,B 0,C 180,E1 12974.841,E2 12974.841} C_VEL
LIN {X 0,Y 410.932,Z 618.302,A -85,B 0,C 180,E1 12971.723,E2 12971.723} C_VEL
LIN {X 0,Y 408.165,Z 613.814,A -85,B 0,C 180,E1 12969.518,E2 12969.518} C_VEL
LIN {X 0,Y 405.742,Z 609.715,A -85,B 0,C 180,E1 12967.078,E2 12967.078} C_VEL
LIN {X 0,Y 403.365,Z 605.282,A -85,B 0,C 180,E1 12963.482,E2 12963.482} C_VEL
LIN {X 0,Y 402.101,Z 604.24,A -85,B 0,C 180,E1 12958.718,E2 12958.718} C_VEL
LIN {X 0,Y 403.348,Z 605.214,A -85,B 0,C 180,E1 12954.024,E2 12954.024} C_VEL
LIN {X 0,Y 405.648,Z 609.558,A -85,B 0,C 180,E1 12950.494,E2 12950.494} C_VEL
LIN {X 0,Y 406.728,Z 611.467,A -85,B 0,C 180,E1 12949.303,E2 12949.303} C_VEL
LIN {X 0,Y 409.188,Z 615.451,A -85,B 0,C 180,E1 12947.08,E2 12947.08} C_VEL
LIN {X 0,Y 412.14,Z 620.424,A -85,B 0,C 180,E1 12944.882,E2 12944.882} C_VEL
LIN {X 0,Y 417.202,Z 630.788,A -85,B 0,C 180,E1 12941.702,E2 12941.702} C_VEL
LIN {X 0,Y 421.307,Z 640.084,A -85,B 0,C 180,E1 12939.496,E2 12939.496} C_VEL
LIN {X 0,Y 404.376,Z 828.493,A -85,B 0,C 180,E1 12936.533,E2 12936.533} C_VEL
LIN {X 0,Y 400.33,Z 855.236,A -85,B 0,C 180,E1 12935.997,E2 12935.997} C_VEL
LIN {X 0,Y 395.794,Z 876.683,A -85,B 0,C 180,E1 12935.454,E2 12935.454} C_VEL
LIN {X 0,Y 389.401,Z 900.795,A -85,B 0,C 180,E1 12934.67,E2 12934.67} C_VEL
LIN {X 0,Y 382.592,Z 921.953,A -85,B 0,C 180,E1 12933.789,E2 12933.789} C_VEL
LIN {X 0,Y 374.4,Z 944.187,A -85,B 0,C 180,E1 12932.639,E2 12932.639} C_VEL
LIN {X 0,Y 365.419,Z 965.127,A -85,B 0,C 180,E1 12931.281,E2 12931.281} C_VEL
LIN {X 0,Y 355.909,Z 985.13,A -85,B 0,C 180,E1 12929.716,E2 12929.716} C_VEL
LIN {X 0,Y 345.163,Z 1005.295,A -85,B 0,C 180,E1 12927.767,E2 12927.767} C_VEL
LIN {X 0,Y 335.117,Z 1022.659,A -85,B 0,C 180,E1 12925.74,E2 12925.74} C_VEL
LIN {X 0,Y 323.661,Z 1040.898,A -85,B 0,C 180,E1 12923.143,E2 12923.143} C_VEL
LIN {X 0,Y 313.51,Z 1056.048,A -85,B 0,C 180,E1 12920.518,E2 12920.518} C_VEL
LIN {X 0,Y 301.951,Z 1072.458,A -85,B 0,C 180,E1 12917.04,E2 12917.04} C_VEL
LIN {X 0,Y 292.504,Z 1085.335,A -85,B 0,C 180,E1 12913.671,E2 12913.671} C_VEL
LIN {X 0,Y 282.856,Z 1098.353,A -85,B 0,C 180,E1 12909.516,E2 12909.516} C_VEL
LIN {X 0,Y 275.016,Z 1108.885,A -85,B 0,C 180,E1 12905.316,E2 12905.316} C_VEL
LIN {X 0,Y 268.042,Z 1118.778,A -85,B 0,C 180,E1 12900.486,E2 12900.486} C_VEL
LIN {X 0,Y 262.756,Z 1126.732,A -85,B 0,C 180,E1 12895.468,E2 12895.468} C_VEL
LIN {X 0,Y 259.261,Z 1132.932,A -85,B 0,C 180,E1 12890.546,E2 12890.546} C_VEL
LIN {X 0,Y 256.966,Z 1138.174,A -85,B 0,C 180,E1 12884.881,E2 12884.881} C_VEL
LIN {X 0,Y 256.174,Z 1141.086,A -85,B 0,C 180,E1 12880.343,E2 12880.343} C_VEL
LIN {X 0,Y 256.014,Z 1142.897,A -85,B 0,C 180,E1 12875.828,E2 12875.828} C_VEL
LIN {X 0,Y 256.081,Z 1143.623,A -85,B 0,C 180,E1 12871.119,E2 12871.119} C_VEL
LIN {X 0,Y 256.056,Z 1143.02,A -85,B 0,C 180,E1 12866.642,E2 12866.642} C_VEL
LIN {X 0,Y 256.03,Z 1141.406,A -85,B 0,C 180,E1 12862.37,E2 12862.37} C_VEL
LIN {X 0,Y 256.352,Z 1138.764,A -85,B 0,C 180,E1 12858.069,E2 12858.069} C_VEL
LIN {X 0,Y 257.462,Z 1134.651,A -85,B 0,C 180,E1 12853.298,E2 12853.298} C_VEL
LIN {X 0,Y 260.22,Z 1127.948,A -85,B 0,C 180,E1 12847.641,E2 12847.641} C_VEL
LIN {X 0,Y 263.927,Z 1120.815,A -85,B 0,C 180,E1 12842.959,E2 12842.959} C_VEL
LIN {X 0,Y 270.159,Z 1110.38,A -85,B 0,C 180,E1 12837.543,E2 12837.543} C_VEL
LIN {X 0,Y 276.583,Z 1100.382,A -85,B 0,C 180,E1 12833.376,E2 12833.376} C_VEL
LIN {X 0,Y 285.5,Z 1086.928,A -85,B 0,C 180,E1 12828.82,E2 12828.82} C_VEL
LIN {X 0,Y 293.918,Z 1074.205,A -85,B 0,C 180,E1 12825.317,E2 12825.317} C_VEL
LIN {X 0,Y 304.175,Z 1058.425,A -85,B 0,C 180,E1 12821.737,E2 12821.737} C_VEL
LIN {X 0,Y 313.635,Z 1043.151,A -85,B 0,C 180,E1 12818.907,E2 12818.907} C_VEL
LIN {X 0,Y 323.938,Z 1025.783,A -85,B 0,C 180,E1 12816.218,E2 12816.218} C_VEL
LIN {X 0,Y 334.145,Z 1007.005,A -85,B 0,C 180,E1 12813.861,E2 12813.861} C_VEL
LIN {X 0,Y 344.129,Z 987.284,A -85,B 0,C 180,E1 12811.801,E2 12811.801} C_VEL
LIN {X 0,Y 353.635,Z 966.242,A -85,B 0,C 180,E1 12810.031,E2 12810.031} C_VEL
LIN {X 0,Y 362.506,Z 944.5,A -85,B 0,C 180,E1 12808.52,E2 12808.52} C_VEL
LIN {X 0,Y 370.21,Z 922.52,A -85,B 0,C 180,E1 12807.303,E2 12807.303} C_VEL
LIN {X 0,Y 376.638,Z 901.603,A -85,B 0,C 180,E1 12806.364,E2 12806.364} C_VEL
LIN {X 0,Y 382.913,Z 876.88,A -85,B 0,C 180,E1 12805.497,E2 12805.497} C_VEL
LIN {X 0,Y 387.243,Z 855.459,A -85,B 0,C 180,E1 12804.915,E2 12804.915} C_VEL
LIN {X 0,Y 391.124,Z 828.354,A -85,B 0,C 180,E1 12804.342,E2 12804.342} C_VEL
LIN {X 0,Y 407.915,Z 630.315,A -85,B 0,C 180,E1 12801.121,E2 12801.121} C_VEL
LIN {X 0,Y 401.776,Z 617.145,A -85,B 0,C 180,E1 12798.275,E2 12798.275} C_VEL
LIN {X 0,Y 396.723,Z 607.112,A -85,B 0,C 180,E1 12795.57,E2 12795.57} C_VEL
LIN {X 0,Y 391.522,Z 598.635,A -85,B 0,C 180,E1 12792.313,E2 12792.313} C_VEL
LIN {X 0,Y 388.171,Z 593.492,A -85,B 0,C 180,E1 12789.714,E2 12789.714} C_VEL
LIN {X 0,Y 385.592,Z 589.289,A -85,B 0,C 180,E1 12787.15,E2 12787.15} C_VEL
LIN {X 0,Y 383.068,Z 585.205,A -85,B 0,C 180,E1 12783.517,E2 12783.517} C_VEL
LIN {X 0,Y 382.708,Z 584.339,A -85,B 0,C 180,E1 12782.695,E2 12782.695} C_VEL
LIN {X 0,Y 381.695,Z 583.721,A -85,B 0,C 180,E1 12777.147,E2 12777.147} C_VEL
LIN {X 0,Y 382.902,Z 584.715,A -85,B 0,C 180,E1 12773.327,E2 12773.327} C_VEL
LIN {X 0,Y 384.991,Z 588.683,A -85,B 0,C 180,E1 12769.979,E2 12769.979} C_VEL
LIN {X 0,Y 386.051,Z 590.058,A -85,B 0,C 180,E1 12768.799,E2 12768.799} C_VEL
LIN {X 0,Y 389.299,Z 595.288,A -85,B 0,C 180,E1 12765.801,E2 12765.801} C_VEL
LIN {X 0,Y 392.449,Z 600.328,A -85,B 0,C 180,E1 12763.496,E2 12763.496} C_VEL
LIN {X 0,Y 396.925,Z 607.577,A -85,B 0,C 180,E1 12760.769,E2 12760.769} C_VEL
LIN {X 0,Y 402.594,Z 617.323,A -85,B 0,C 180,E1 12757.859,E2 12757.859} C_VEL
LIN {X 0,Y 408.062,Z 627.188,A -85,B 0,C 180,E1 12755.43,E2 12755.43} C_VEL
LIN {X 0,Y 391.831,Z 817.099,A -85,B 0,C 180,E1 12752.361,E2 12752.361} C_VEL
LIN {X 0,Y 388.066,Z 843.546,A -85,B 0,C 180,E1 12751.775,E2 12751.775} C_VEL
LIN {X 0,Y 384.036,Z 864.268,A -85,B 0,C 180,E1 12751.16,E2 12751.16} C_VEL
LIN {X 0,Y 378.137,Z 888.49,A -85,B 0,C 180,E1 12750.244,E2 12750.244} C_VEL
LIN {X 0,Y 371.813,Z 909.692,A -85,B 0,C 180,E1 12749.228,E2 12749.228} C_VEL
LIN {X 0,Y 364.089,Z 932.156,A -85,B 0,C 180,E1 12747.912,E2 12747.912} C_VEL
LIN {X 0,Y 355.812,Z 952.691,A -85,B 0,C 180,E1 12746.431,E2 12746.431} C_VEL
LIN {X 0,Y 346.822,Z 972.9,A -85,B 0,C 180,E1 12744.676,E2 12744.676} C_VEL
LIN {X 0,Y 337.155,Z 992.148,A -85,B 0,C 180,E1 12742.637,E2 12742.637} C_VEL
LIN {X 0,Y 327.616,Z 1009.709,A -85,B 0,C 180,E1 12740.411,E2 12740.411} C_VEL
LIN {X 0,Y 317.416,Z 1026.98,A -85,B 0,C 180,E1 12737.755,E2 12737.755} C_VEL
LIN {X 0,Y 308.145,Z 1041.745,A -85,B 0,C 180,E1 12735.023,E2 12735.023} C_VEL
LIN {X 0,Y 297.633,Z 1057.682,A -85,B 0,C 180,E1 12731.439,E2 12731.439} C_VEL
LIN {X 0,Y 289.06,Z 1070.151,A -85,B 0,C 180,E1 12728.005,E2 12728.005} C_VEL
LIN {X 0,Y 280.353,Z 1082.714,A -85,B 0,C 180,E1 12723.798,E2 12723.798} C_VEL
LIN {X 0,Y 273.327,Z 1092.796,A -85,B 0,C 180,E1 12719.595,E2 12719.595} C_VEL
LIN {X 0,Y 267.108,Z 1102.226,A -85,B 0,C 180,E1 12714.788,E2 12714.788} C_VEL
LIN {X 0,Y 262.302,Z 1109.942,A -85,B 0,C 180,E1 12709.684,E2 12709.684} C_VEL
LIN {X 0,Y 259.083,Z 1116.078,A -85,B 0,C 180,E1 12704.528,E2 12704.528} C_VEL
LIN {X 0,Y 257.131,Z 1120.603,A -85,B 0,C 180,E1 12699.174,E2 12699.174} C_VEL
LIN {X 0,Y 256.376,Z 1123.233,A -85,B 0,C 180,E1 12694.698,E2 12694.698} C_VEL
LIN {X 0,Y 256.136,Z 1124.901,A -85,B 0,C 180,E1 12690,E2 12690} C_VEL
LIN {X 0,Y 256.095,Z 1125.343,A -85,B 0,C 180,E1 12685.072,E2 12685.072} C_VEL
LIN {X 0,Y 256.31,Z 1124.636,A -85,B 0,C 180,E1 12680.57,E2 12680.57} C_VEL
LIN {X 0,Y 256.884,Z 1123.008,A -85,B 0,C 180,E1 12676.265,E2 12676.265} C_VEL
LIN {X 0,Y 258.503,Z 1119.798,A -85,B 0,C 180,E1 12671.04,E2 12671.04} C_VEL
LIN {X 0,Y 261.581,Z 1114.676,A -85,B 0,C 180,E1 12665.617,E2 12665.617} C_VEL
LIN {X 0,Y 265.876,Z 1108.585,A -85,B 0,C 180,E1 12660.732,E2 12660.732} C_VEL
LIN {X 0,Y 272.251,Z 1100.096,A -85,B 0,C 180,E1 12655.556,E2 12655.556} C_VEL
LIN {X 0,Y 279.317,Z 1091.103,A -85,B 0,C 180,E1 12651.21,E2 12651.21} C_VEL
LIN {X 0,Y 288.6,Z 1079.305,A -85,B 0,C 180,E1 12646.683,E2 12646.683} C_VEL
LIN {X 0,Y 297.422,Z 1067.931,A -85,B 0,C 180,E1 12643.153,E2 12643.153} C_VEL
LIN {X 0,Y 308.876,Z 1052.62,A -85,B 0,C 180,E1 12639.313,E2 12639.313} C_VEL
LIN {X 0,Y 318.554,Z 1038.982,A -85,B 0,C 180,E1 12636.53,E2 12636.53} C_VEL
LIN {X 0,Y 330.163,Z 1021.604,A -85,B 0,C 180,E1 12633.609,E2 12633.609} C_VEL
LIN {X 0,Y 339.862,Z 1005.865,A -85,B 0,C 180,E1 12631.439,E2 12631.439} C_VEL
LIN {X 0,Y 350.321,Z 987.635,A -85,B 0,C 180,E1 12629.329,E2 12629.329} C_VEL
LIN {X 0,Y 360.173,Z 968.366,A -85,B 0,C 180,E1 12627.504,E2 12627.504} C_VEL
LIN {X 0,Y 368.526,Z 950.404,A -85,B 0,C 180,E1 12626.075,E2 12626.075} C_VEL
LIN {X 0,Y 378.143,Z 926.948,A -85,B 0,C 180,E1 12624.548,E2 12624.548} C_VEL
LIN {X 0,Y 384.941,Z 907.75,A -85,B 0,C 180,E1 12623.519,E2 12623.519} C_VEL
LIN {X 0,Y 392.126,Z 884.106,A -85,B 0,C 180,E1 12622.488,E2 12622.488} C_VEL
LIN {X 0,Y 397.595,Z 861.858,A -85,B 0,C 180,E1 12621.731,E2 12621.731} C_VEL
LIN {X 0,Y 402.272,Z 838.132,A -85,B 0,C 180,E1 12621.099,E2 12621.099} C_VEL
LIN {X 0,Y 405.513,Z 813.99,A -85,B 0,C 180,E1 12620.625,E2 12620.625} C_VEL
LIN {X 0,Y 416.828,Z 687.998,A -85,B 0,C 180,E1 12618.644,E2 12618.644} C_VEL
LIN {X 0,Y 417.172,Z 680.448,A -85,B 0,C 180,E1 12618.399,E2 12618.399} C_VEL
LIN {X 0,Y 416.908,Z 660.804,A -85,B 0,C 180,E1 12617.287,E2 12617.287} C_VEL
LIN {X 0,Y 417.264,Z 654.312,A -85,B 0,C 180,E1 12617.088,E2 12617.088} C_VEL
LIN {X 0,Y 418.377,Z 641.848,A -85,B 0,C 180,E1 12616.881,E2 12616.881} C_VEL
LIN {X 0,Y 413.517,Z 633.029,A -85,B 0,C 180,E1 12614.157,E2 12614.157} C_VEL
LIN {X 0,Y 409.467,Z 625.849,A -85,B 0,C 180,E1 12611.408,E2 12611.408} C_VEL
LIN {X 0,Y 406.783,Z 621.397,A -85,B 0,C 180,E1 12609.194,E2 12609.194} C_VEL
LIN {X 0,Y 404.511,Z 617.456,A -85,B 0,C 180,E1 12606.814,E2 12606.814} C_VEL
LIN {X 0,Y 402.148,Z 612.958,A -85,B 0,C 180,E1 12602.993,E2 12602.993} C_VEL
LIN {X 0,Y 401.156,Z 612.199,A -85,B 0,C 180,E1 12598,E2 12598} C_VEL
LIN {X 0,Y 402.327,Z 613.237,A -85,B 0,C 180,E1 12594.08,E2 12594.08} C_VEL
LIN {X 0,Y 404.677,Z 617.575,A -85,B 0,C 180,E1 12590.471,E2 12590.471} C_VEL
LIN {X 0,Y 407.784,Z 623,A -85,B 0,C 180,E1 12587.395,E2 12587.395} C_VEL
LIN {X 0,Y 410.647,Z 628,A -85,B 0,C 180,E1 12585.187,E2 12585.187} C_VEL
LIN {X 0,Y 415.408,Z 638.065,A -85,B 0,C 180,E1 12582.092,E2 12582.092} C_VEL
LIN {X 0,Y 418.291,Z 644.799,A -85,B 0,C 180,E1 12580.459,E2 12580.459} C_VEL
LIN {X 0,Y 401.415,Z 828.331,A -85,B 0,C 180,E1 12577.595,E2 12577.595} C_VEL
LIN {X 0,Y 397.319,Z 854.917,A -85,B 0,C 180,E1 12577.069,E2 12577.069} C_VEL
LIN {X 0,Y 392.691,Z 876.443,A -85,B 0,C 180,E1 12576.533,E2 12576.533} C_VEL
LIN {X 0,Y 386.038,Z 901.023,A -85,B 0,C 180,E1 12575.746,E2 12575.746} C_VEL
LIN {X 0,Y 379.009,Z 922.411,A -85,B 0,C 180,E1 12574.865,E2 12574.865} C_VEL
LIN {X 0,Y 370.338,Z 945.251,A -85,B 0,C 180,E1 12573.687,E2 12573.687} C_VEL
LIN {X 0,Y 361.68,Z 964.999,A -85,B 0,C 180,E1 12572.416,E2 12572.416} C_VEL
LIN {X 0,Y 351.981,Z 984.948,A -85,B 0,C 180,E1 12570.872,E2 12570.872} C_VEL
LIN {X 0,Y 340.888,Z 1005.248,A -85,B 0,C 180,E1 12568.926,E2 12568.926} C_VEL
LIN {X 0,Y 330.586,Z 1022.59,A -85,B 0,C 180,E1 12566.911,E2 12566.911} C_VEL
LIN {X 0,Y 318.703,Z 1040.944,A -85,B 0,C 180,E1 12564.299,E2 12564.299} C_VEL
LIN {X 0,Y 308.342,Z 1055.925,A -85,B 0,C 180,E1 12561.699,E2 12561.699} C_VEL
LIN {X 0,Y 296.382,Z 1072.304,A -85,B 0,C 180,E1 12558.209,E2 12558.209} C_VEL
LIN {X 0,Y 286.568,Z 1085.167,A -85,B 0,C 180,E1 12554.815,E2 12554.815} C_VEL
LIN {X 0,Y 276.422,Z 1098.269,A -85,B 0,C 180,E1 12550.569,E2 12550.569} C_VEL
LIN {X 0,Y 268.289,Z 1108.682,A -85,B 0,C 180,E1 12546.34,E2 12546.34} C_VEL
LIN {X 0,Y 260.937,Z 1118.557,A -85,B 0,C 180,E1 12541.409,E2 12541.409} C_VEL
LIN {X 0,Y 255.313,Z 1126.513,A -85,B 0,C 180,E1 12536.254,E2 12536.254} C_VEL
LIN {X 0,Y 251.576,Z 1132.689,A -85,B 0,C 180,E1 12531.204,E2 12531.204} C_VEL
LIN {X 0,Y 249.083,Z 1137.914,A -85,B 0,C 180,E1 12525.364,E2 12525.364} C_VEL
LIN {X 0,Y 248.196,Z 1140.868,A -85,B 0,C 180,E1 12520.583,E2 12520.583} C_VEL
LIN {X 0,Y 248.015,Z 1142.696,A -85,B 0,C 180,E1 12515.785,E2 12515.785} C_VEL
LIN {X 0,Y 248.085,Z 1143.318,A -85,B 0,C 180,E1 12510.924,E2 12510.924} C_VEL
LIN {X 0,Y 248.061,Z 1142.722,A -85,B 0,C 180,E1 12506.534,E2 12506.534} C_VEL
LIN {X 0,Y 248.039,Z 1141.097,A -85,B 0,C 180,E1 12502.122,E2 12502.122} C_VEL
LIN {X 0,Y 248.4,Z 1138.443,A -85,B 0,C 180,E1 12497.682,E2 12497.682} C_VEL
LIN {X 0,Y 249.629,Z 1134.319,A -85,B 0,C 180,E1 12492.758,E2 12492.758} C_VEL
LIN {X 0,Y 252.454,Z 1127.908,A -85,B 0,C 180,E1 12487.161,E2 12487.161} C_VEL
LIN {X 0,Y 256.351,Z 1120.815,A -85,B 0,C 180,E1 12482.344,E2 12482.344} C_VEL
LIN {X 0,Y 262.578,Z 1110.936,A -85,B 0,C 180,E1 12477.007,E2 12477.007} C_VEL
LIN {X 0,Y 269.207,Z 1101.049,A -85,B 0,C 180,E1 12472.741,E2 12472.741} C_VEL
LIN {X 0,Y 277.549,Z 1089.096,A -85,B 0,C 180,E1 12468.48,E2 12468.48} C_VEL
LIN {X 0,Y 286.731,Z 1075.703,A -85,B 0,C 180,E1 12464.652,E2 12464.652} C_VEL
LIN {X 0,Y 296.529,Z 1061.284,A -85,B 0,C 180,E1 12461.24,E2 12461.24} C_VEL
LIN {X 0,Y 307.265,Z 1044.64,A -85,B 0,C 180,E1 12458.046,E2 12458.046} C_VEL
LIN {X 0,Y 316.997,Z 1028.78,A -85,B 0,C 180,E1 12455.531,E2 12455.531} C_VEL
LIN {X 0,Y 328.296,Z 1008.94,A -85,B 0,C 180,E1 12452.955,E2 12452.955} C_VEL
LIN {X 0,Y 337.438,Z 991.472,A -85,B 0,C 180,E1 12451.089,E2 12451.089} C_VEL
LIN {X 0,Y 347.673,Z 970.057,A -85,B 0,C 180,E1 12449.208,E2 12449.208} C_VEL
LIN {X 0,Y 356.048,Z 950.326,A -85,B 0,C 180,E1 12447.795,E2 12447.795} C_VEL
LIN {X 0,Y 364.284,Z 928.642,A -85,B 0,C 180,E1 12446.516,E2 12446.516} C_VEL
LIN {X 0,Y 371.159,Z 907.29,A -85,B 0,C 180,E1 12445.513,E2 12445.513} C_VEL
LIN {X 0,Y 376.997,Z 886.256,A -85,B 0,C 180,E1 12444.715,E2 12444.715} C_VEL
LIN {X 0,Y 382.735,Z 860.549,A -85,B 0,C 180,E1 12443.97,E2 12443.97} C_VEL
LIN {X 0,Y 386.428,Z 838.305,A -85,B 0,C 180,E1 12443.47,E2 12443.47} C_VEL
LIN {X 0,Y 389.821,Z 805.568,A -85,B 0,C 180,E1 12442.892,E2 12442.892} C_VEL
LIN {X 0,Y 404.475,Z 634.627,A -85,B 0,C 180,E1 12440.135,E2 12440.135} C_VEL
LIN {X 0,Y 398.765,Z 622.189,A -85,B 0,C 180,E1 12437.323,E2 12437.323} C_VEL
LIN {X 0,Y 394.725,Z 614.086,A -85,B 0,C 180,E1 12435.049,E2 12435.049} C_VEL
LIN {X 0,Y 389.913,Z 606.052,A -85,B 0,C 180,E1 12431.913,E2 12431.913} C_VEL
LIN {X 0,Y 386.763,Z 601.071,A -85,B 0,C 180,E1 12429.374,E2 12429.374} C_VEL
LIN {X 0,Y 384.343,Z 597.036,A -85,B 0,C 180,E1 12426.873,E2 12426.873} C_VEL
LIN {X 0,Y 381.916,Z 592.79,A -85,B 0,C 180,E1 12423.152,E2 12423.152} C_VEL
LIN {X 0,Y 381.525,Z 592.175,A -85,B 0,C 180,E1 12422.253,E2 12422.253} C_VEL
LIN {X 0,Y 380.76,Z 591.7,A -85,B 0,C 180,E1 12416.839,E2 12416.839} C_VEL
LIN {X 0,Y 381.823,Z 592.525,A -85,B 0,C 180,E1 12413.534,E2 12413.534} C_VEL
LIN {X 0,Y 383.894,Z 596.566,A -85,B 0,C 180,E1 12410.101,E2 12410.101} C_VEL
LIN {X 0,Y 384.927,Z 598.035,A -85,B 0,C 180,E1 12408.917,E2 12408.917} C_VEL
LIN {X 0,Y 387.955,Z 602.999,A -85,B 0,C 180,E1 12406.055,E2 12406.055} C_VEL
LIN {X 0,Y 390.931,Z 607.884,A -85,B 0,C 180,E1 12403.812,E2 12403.812} C_VEL
LIN {X 0,Y 395.191,Z 614.98,A -85,B 0,C 180,E1 12401.134,E2 12401.134} C_VEL
LIN {X 0,Y 400.933,Z 625.089,A -85,B 0,C 180,E1 12398.109,E2 12398.109} C_VEL
LIN {X 0,Y 404.608,Z 632.056,A -85,B 0,C 180,E1 12396.399,E2 12396.399} C_VEL
LIN {X 0,Y 388.383,Z 817.417,A -85,B 0,C 180,E1 12393.421,E2 12393.421} C_VEL
LIN {X 0,Y 384.526,Z 843.947,A -85,B 0,C 180,E1 12392.838,E2 12392.838} C_VEL
LIN {X 0,Y 380.432,Z 864.574,A -85,B 0,C 180,E1 12392.232,E2 12392.232} C_VEL
LIN {X 0,Y 374.382,Z 888.902,A -85,B 0,C 180,E1 12391.32,E2 12391.32} C_VEL
LIN {X 0,Y 368.162,Z 909.368,A -85,B 0,C 180,E1 12390.353,E2 12390.353} C_VEL
LIN {X 0,Y 360.624,Z 931.003,A -85,B 0,C 180,E1 12389.109,E2 12389.109} C_VEL
LIN {X 0,Y 351.8,Z 952.541,A -85,B 0,C 180,E1 12387.58,E2 12387.58} C_VEL
LIN {X 0,Y 342.919,Z 972.069,A -85,B 0,C 180,E1 12385.904,E2 12385.904} C_VEL
LIN {X 0,Y 332.561,Z 992.3,A -85,B 0,C 180,E1 12383.785,E2 12383.785} C_VEL
LIN {X 0,Y 323.141,Z 1009.19,A -85,B 0,C 180,E1 12381.657,E2 12381.657} C_VEL
LIN {X 0,Y 312.045,Z 1027.479,A -85,B 0,C 180,E1 12378.853,E2 12378.853} C_VEL
LIN {X 0,Y 302.481,Z 1042.226,A -85,B 0,C 180,E1 12376.107,E2 12376.107} C_VEL
LIN {X 0,Y 291.611,Z 1058.13,A -85,B 0,C 180,E1 12372.492,E2 12372.492} C_VEL
LIN {X 0,Y 282.714,Z 1070.585,A -85,B 0,C 180,E1 12369.017,E2 12369.017} C_VEL
LIN {X 0,Y 273.442,Z 1083.386,A -85,B 0,C 180,E1 12364.638,E2 12364.638} C_VEL
LIN {X 0,Y 266.302,Z 1093.191,A -85,B 0,C 180,E1 12360.457,E2 12360.457} C_VEL
LIN {X 0,Y 259.77,Z 1102.599,A -85,B 0,C 180,E1 12355.538,E2 12355.538} C_VEL
LIN {X 0,Y 254.815,Z 1110.112,A -85,B 0,C 180,E1 12350.441,E2 12350.441} C_VEL
LIN {X 0,Y 251.399,Z 1116.176,A -85,B 0,C 180,E1 12345.219,E2 12345.219} C_VEL
LIN {X 0,Y 249.267,Z 1120.771,A -85,B 0,C 180,E1 12339.699,E2 12339.699} C_VEL
LIN {X 0,Y 248.427,Z 1123.434,A -85,B 0,C 180,E1 12335.08,E2 12335.08} C_VEL
LIN {X 0,Y 248.151,Z 1125.134,A -85,B 0,C 180,E1 12330.231,E2 12330.231} C_VEL
LIN {X 0,Y 248.1,Z 1125.645,A -85,B 0,C 180,E1 12325.145,E2 12325.145} C_VEL
LIN {X 0,Y 248.321,Z 1124.973,A -85,B 0,C 180,E1 12320.497,E2 12320.497} C_VEL
LIN {X 0,Y 248.982,Z 1123.271,A -85,B 0,C 180,E1 12315.82,E2 12315.82} C_VEL
LIN {X 0,Y 250.749,Z 1120.052,A -85,B 0,C 180,E1 12310.43,E2 12310.43} C_VEL
LIN {X 0,Y 254.087,Z 1114.899,A -85,B 0,C 180,E1 12304.838,E2 12304.838} C_VEL
LIN {X 0,Y 258.905,Z 1108.513,A -85,B 0,C 180,E1 12299.607,E2 12299.607} C_VEL
LIN {X 0,Y 265.637,Z 1100.031,A -85,B 0,C 180,E1 12294.396,E2 12294.396} C_VEL
LIN {X 0,Y 273.373,Z 1090.721,A -85,B 0,C 180,E1 12289.858,E2 12289.858} C_VEL
LIN {X 0,Y 282.598,Z 1079.471,A -85,B 0,C 180,E1 12285.527,E2 12285.527} C_VEL
LIN {X 0,Y 291.994,Z 1067.839,A -85,B 0,C 180,E1 12281.894,E2 12281.894} C_VEL
LIN {X 0,Y 303.691,Z 1052.735,A -85,B 0,C 180,E1 12278.103,E2 12278.103} C_VEL
LIN {X 0,Y 313.7,Z 1039.081,A -85,B 0,C 180,E1 12275.316,E2 12275.316} C_VEL
LIN {X 0,Y 325.988,Z 1021.157,A -85,B 0,C 180,E1 12272.324,E2 12272.324} C_VEL
LIN {X 0,Y 335.742,Z 1005.74,A -85,B 0,C 180,E1 12270.219,E2 12270.219} C_VEL
LIN {X 0,Y 346.765,Z 986.921,A -85,B 0,C 180,E1 12268.073,E2 12268.073} C_VEL
LIN {X 0,Y 356.832,Z 967.584,A -85,B 0,C 180,E1 12266.274,E2 12266.274} C_VEL
LIN {X 0,Y 366.109,Z 947.97,A -85,B 0,C 180,E1 12264.755,E2 12264.755} C_VEL
LIN {X 0,Y 374.835,Z 926.782,A -85,B 0,C 180,E1 12263.416,E2 12263.416} C_VEL
LIN {X 0,Y 382.163,Z 906.392,A -85,B 0,C 180,E1 12262.347,E2 12262.347} C_VEL
LIN {X 0,Y 389.606,Z 881.779,A -85,B 0,C 180,E1 12261.312,E2 12261.312} C_VEL
LIN {X 0,Y 394.942,Z 860.148,A -85,B 0,C 180,E1 12260.601,E2 12260.601} C_VEL
LIN {X 0,Y 399.911,Z 833.965,A -85,B 0,C 180,E1 12259.943,E2 12259.943} C_VEL
LIN {X 0,Y 402.822,Z 811.857,A -85,B 0,C 180,E1 12259.529,E2 12259.529} C_VEL
LIN {X 0,Y 417.264,Z 654.312,A -85,B 0,C 180,E1 12257.088,E2 12257.088} C_VEL
LIN {X 0,Y 417.239,Z 651.081,A -85,B 0,C 180,E1 12256.904,E2 12256.904} C_VEL
LIN {X 0,Y 416.607,Z 648.098,A -85,B 0,C 180,E1 12256.474,E2 12256.474} C_VEL
LIN {X 0,Y 415.221,Z 645.449,A -85,B 0,C 180,E1 12255.717,E2 12255.717} C_VEL
LIN {X 0,Y 412.711,Z 641.922,A -85,B 0,C 180,E1 12254.32,E2 12254.32} C_VEL
LIN {X 0,Y 408.197,Z 633.667,A -85,B 0,C 180,E1 12251.229,E2 12251.229} C_VEL
LIN {X 0,Y 405.49,Z 629.086,A -85,B 0,C 180,E1 12248.937,E2 12248.937} C_VEL
LIN {X 0,Y 403.41,Z 625.331,A -85,B 0,C 180,E1 12246.69,E2 12246.69} C_VEL
LIN {X 0,Y 401.105,Z 620.863,A -85,B 0,C 180,E1 12242.858,E2 12242.858} C_VEL
LIN {X 0,Y 400.181,Z 620.14,A -85,B 0,C 180,E1 12237.995,E2 12237.995} C_VEL
LIN {X 0,Y 401.28,Z 621.148,A -85,B 0,C 180,E1 12234.208,E2 12234.208} C_VEL
LIN {X 0,Y 403.926,Z 626.197,A -85,B 0,C 180,E1 12230.165,E2 12230.165} C_VEL
LIN {X 0,Y 406.626,Z 631.016,A -85,B 0,C 180,E1 12227.503,E2 12227.503} C_VEL
LIN {X 0,Y 409.166,Z 635.574,A -85,B 0,C 180,E1 12225.494,E2 12225.494} C_VEL
LIN {X 0,Y 413.688,Z 645.468,A -85,B 0,C 180,E1 12222.451,E2 12222.451} C_VEL
LIN {X 0,Y 415.369,Z 649.781,A -85,B 0,C 180,E1 12221.432,E2 12221.432} C_VEL
LIN {X 0,Y 398.618,Z 827.978,A -85,B 0,C 180,E1 12218.675,E2 12218.675} C_VEL
LIN {X 0,Y 394.426,Z 854.721,A -85,B 0,C 180,E1 12218.153,E2 12218.153} C_VEL
LIN {X 0,Y 389.705,Z 876.312,A -85,B 0,C 180,E1 12217.627,E2 12217.627} C_VEL
LIN {X 0,Y 382.815,Z 901.25,A -85,B 0,C 180,E1 12216.84,E2 12216.84} C_VEL
LIN {X 0,Y 375.939,Z 921.806,A -85,B 0,C 180,E1 12216.01,E2 12216.01} C_VEL
LIN {X 0,Y 367.171,Z 944.558,A -85,B 0,C 180,E1 12214.86,E2 12214.86} C_VEL
LIN {X 0,Y 358.314,Z 964.392,A -85,B 0,C 180,E1 12213.607,E2 12213.607} C_VEL
LIN {X 0,Y 348.702,Z 983.778,A -85,B 0,C 180,E1 12212.134,E2 12212.134} C_VEL
LIN {X 0,Y 337.476,Z 1003.985,A -85,B 0,C 180,E1 12210.241,E2 12210.241} C_VEL
LIN {X 0,Y 327.578,Z 1020.296,A -85,B 0,C 180,E1 12208.388,E2 12208.388} C_VEL
LIN {X 0,Y 315.409,Z 1038.825,A -85,B 0,C 180,E1 12205.834,E2 12205.834} C_VEL
LIN {X 0,Y 304.547,Z 1054.101,A -85,B 0,C 180,E1 12203.236,E2 12203.236} C_VEL
LIN {X 0,Y 293.225,Z 1069.298,A -85,B 0,C 180,E1 12200.108,E2 12200.108} C_VEL
LIN {X 0,Y 282.297,Z 1083.076,A -85,B 0,C 180,E1 12196.561,E2 12196.561} C_VEL
LIN {X 0,Y 272.524,Z 1095.191,A -85,B 0,C 180,E1 12192.748,E2 12192.748} C_VEL
LIN {X 0,Y 262.745,Z 1107.141,A -85,B 0,C 180,E1 12188.024,E2 12188.024} C_VEL
LIN {X 0,Y 255.425,Z 1116.29,A -85,B 0,C 180,E1 12183.502,E2 12183.502} C_VEL
LIN {X 0,Y 248.54,Z 1125.425,A -85,B 0,C 180,E1 12177.739,E2 12177.739} C_VEL
LIN {X 0,Y 244.376,Z 1131.66,A -85,B 0,C 180,E1 12172.62,E2 12172.62} C_VEL
LIN {X 0,Y 241.435,Z 1137.153,A -85,B 0,C 180,E1 12166.604,E2 12166.604} C_VEL
LIN {X 0,Y 240.296,Z 1140.312,A -85,B 0,C 180,E1 12161.521,E2 12161.521} C_VEL
LIN {X 0,Y 240.033,Z 1142.133,A -85,B 0,C 180,E1 12156.939,E2 12156.939} C_VEL
LIN {X 0,Y 240.066,Z 1142.946,A -85,B 0,C 180,E1 12152.387,E2 12152.387} C_VEL
LIN {X 0,Y 240.081,Z 1142.738,A -85,B 0,C 180,E1 12147.852,E2 12147.852} C_VEL
LIN {X 0,Y 240.037,Z 1141.26,A -85,B 0,C 180,E1 12142.821,E2 12142.821} C_VEL
LIN {X 0,Y 240.387,Z 1138.456,A -85,B 0,C 180,E1 12137.752,E2 12137.752} C_VEL
LIN {X 0,Y 241.547,Z 1134.632,A -85,B 0,C 180,E1 12132.908,E2 12132.908} C_VEL
LIN {X 0,Y 244.389,Z 1128.495,A -85,B 0,C 180,E1 12127.127,E2 12127.127} C_VEL
LIN {X 0,Y 248.576,Z 1121.18,A -85,B 0,C 180,E1 12121.925,E2 12121.925} C_VEL
LIN {X 0,Y 254.713,Z 1111.961,A -85,B 0,C 180,E1 12116.662,E2 12116.662} C_VEL
LIN {X 0,Y 262.248,Z 1101.178,A -85,B 0,C 180,E1 12111.854,E2 12111.854} C_VEL
LIN {X 0,Y 270.923,Z 1089.278,A -85,B 0,C 180,E1 12107.515,E2 12107.515} C_VEL
LIN {X 0,Y 280.95,Z 1075.267,A -85,B 0,C 180,E1 12103.445,E2 12103.445} C_VEL
LIN {X 0,Y 291.459,Z 1060.36,A -85,B 0,C 180,E1 12099.906,E2 12099.906} C_VEL
LIN {X 0,Y 302.402,Z 1043.882,A -85,B 0,C 180,E1 12096.761,E2 12096.761} C_VEL
LIN {X 0,Y 312.586,Z 1027.764,A -85,B 0,C 180,E1 12094.22,E2 12094.22} C_VEL
LIN {X 0,Y 323.739,Z 1008.664,A -85,B 0,C 180,E1 12091.762,E2 12091.762} C_VEL
LIN {X 0,Y 333.349,Z 990.752,A -85,B 0,C 180,E1 12089.863,E2 12089.863} C_VEL
LIN {X 0,Y 344.115,Z 968.616,A -85,B 0,C 180,E1 12087.953,E2 12087.953} C_VEL
LIN {X 0,Y 352.687,Z 948.759,A -85,B 0,C 180,E1 12086.56,E2 12086.56} C_VEL
LIN {X 0,Y 361.486,Z 925.606,A -85,B 0,C 180,E1 12085.243,E2 12085.243} C_VEL
LIN {X 0,Y 368.13,Z 905.183,A -85,B 0,C 180,E1 12084.319,E2 12084.319} C_VEL
LIN {X 0,Y 374.497,Z 882.383,A -85,B 0,C 180,E1 12083.489,E2 12083.489} C_VEL
LIN {X 0,Y 379.735,Z 858.289,A -85,B 0,C 180,E1 12082.827,E2 12082.827} C_VEL
LIN {X 0,Y 383.665,Z 834.314,A -85,B 0,C 180,E1 12082.303,E2 12082.303} C_VEL
LIN {X 0,Y 387.532,Z 794.349,A -85,B 0,C 180,E1 12081.632,E2 12081.632} C_VEL
LIN {X 0,Y 401.149,Z 639.16,A -85,B 0,C 180,E1 12079.141,E2 12079.141} C_VEL
LIN {X 0,Y 396.48,Z 628.657,A -85,B 0,C 180,E1 12076.708,E2 12076.708} C_VEL
LIN {X 0,Y 392.877,Z 621.256,A -85,B 0,C 180,E1 12074.594,E2 12074.594} C_VEL
LIN {X 0,Y 388.423,Z 613.599,A -85,B 0,C 180,E1 12071.583,E2 12071.583} C_VEL
LIN {X 0,Y 385.37,Z 608.648,A -85,B 0,C 180,E1 12069.031,E2 12069.031} C_VEL
LIN {X 0,Y 383.104,Z 604.777,A -85,B 0,C 180,E1 12066.594,E2 12066.594} C_VEL
LIN {X 0,Y 380.806,Z 600.479,A -85,B 0,C 180,E1 12062.86,E2 12062.86} C_VEL
LIN {X 0,Y 379.686,Z 599.561,A -85,B 0,C 180,E1 12058.491,E2 12058.491} C_VEL
LIN {X 0,Y 380.776,Z 600.445,A -85,B 0,C 180,E1 12053.668,E2 12053.668} C_VEL
LIN {X 0,Y 382.924,Z 604.585,A -85,B 0,C 180,E1 12050.076,E2 12050.076} C_VEL
LIN {X 0,Y 383.805,Z 606.006,A -85,B 0,C 180,E1 12049.037,E2 12049.037} C_VEL
LIN {X 0,Y 386.619,Z 610.708,A -85,B 0,C 180,E1 12046.312,E2 12046.312} C_VEL
LIN {X 0,Y 389.525,Z 615.618,A -85,B 0,C 180,E1 12044.058,E2 12044.058} C_VEL
LIN {X 0,Y 393.687,Z 622.784,A -85,B 0,C 180,E1 12041.374,E2 12041.374} C_VEL
LIN {X 0,Y 399.35,Z 632.985,A -85,B 0,C 180,E1 12038.327,E2 12038.327} C_VEL
LIN {X 0,Y 401.266,Z 636.942,A -85,B 0,C 180,E1 12037.385,E2 12037.385} C_VEL
LIN {X 0,Y 385.071,Z 817.735,A -85,B 0,C 180,E1 12034.499,E2 12034.499} C_VEL
LIN {X 0,Y 381.162,Z 844.122,A -85,B 0,C 180,E1 12033.926,E2 12033.926} C_VEL
LIN {X 0,Y 376.988,Z 864.767,A -85,B 0,C 180,E1 12033.327,E2 12033.327} C_VEL
LIN {X 0,Y 371.017,Z 888.451,A -85,B 0,C 180,E1 12032.456,E2 12032.456} C_VEL
LIN {X 0,Y 364.288,Z 910.153,A -85,B 0,C 180,E1 12031.442,E2 12031.442} C_VEL
LIN {X 0,Y 356.23,Z 932.642,A -85,B 0,C 180,E1 12030.15,E2 12030.15} C_VEL
LIN {X 0,Y 347.578,Z 953.189,A -85,B 0,C 180,E1 12028.693,E2 12028.693} C_VEL
LIN {X 0,Y 338.149,Z 973.408,A -85,B 0,C 180,E1 12026.961,E2 12026.961} C_VEL
LIN {X 0,Y 327.651,Z 993.268,A -85,B 0,C 180,E1 12024.871,E2 12024.871} C_VEL
LIN {X 0,Y 317.28,Z 1011.329,A -85,B 0,C 180,E1 12022.577,E2 12022.577} C_VEL
LIN {X 0,Y 306.195,Z 1028.884,A -85,B 0,C 180,E1 12019.83,E2 12019.83} C_VEL
LIN {X 0,Y 296.18,Z 1043.825,A -85,B 0,C 180,E1 12017.004,E2 12017.004} C_VEL
LIN {X 0,Y 285.178,Z 1059.265,A -85,B 0,C 180,E1 12013.41,E2 12013.41} C_VEL
LIN {X 0,Y 276.462,Z 1071.019,A -85,B 0,C 180,E1 12010.075,E2 12010.075} C_VEL
LIN {X 0,Y 266.595,Z 1084.055,A -85,B 0,C 180,E1 12005.523,E2 12005.523} C_VEL
LIN {X 0,Y 259.007,Z 1094.032,A -85,B 0,C 180,E1 12001.152,E2 12001.152} C_VEL
LIN {X 0,Y 251.952,Z 1103.655,A -85,B 0,C 180,E1 11995.884,E2 11995.884} C_VEL
LIN {X 0,Y 247.057,Z 1110.764,A -85,B 0,C 180,E1 11990.864,E2 11990.864} C_VEL
LIN {X 0,Y 243.38,Z 1116.987,A -85,B 0,C 180,E1 11985.244,E2 11985.244} C_VEL
LIN {X 0,Y 241.286,Z 1121.247,A -85,B 0,C 180,E1 11979.782,E2 11979.782} C_VEL
LIN {X 0,Y 240.423,Z 1123.854,A -85,B 0,C 180,E1 11975.01,E2 11975.01} C_VEL
LIN {X 0,Y 240.135,Z 1125.568,A -85,B 0,C 180,E1 11969.761,E2 11969.761} C_VEL
LIN {X 0,Y 240.124,Z 1125.883,A -85,B 0,C 180,E1 11964.504,E2 11964.504} C_VEL
LIN {X 0,Y 240.364,Z 1125.181,A -85,B 0,C 180,E1 11959.938,E2 11959.938} C_VEL
LIN {X 0,Y 241.09,Z 1123.535,A -85,B 0,C 180,E1 11955.345,E2 11955.345} C_VEL
LIN {X 0,Y 243.063,Z 1120.248,A -85,B 0,C 180,E1 11949.707,E2 11949.707} C_VEL
LIN {X 0,Y 246.62,Z 1115.144,A -85,B 0,C 180,E1 11944.032,E2 11944.032} C_VEL
LIN {X 0,Y 251.816,Z 1108.693,A -85,B 0,C 180,E1 11938.618,E2 11938.618} C_VEL
LIN {X 0,Y 258.689,Z 1100.497,A -85,B 0,C 180,E1 11933.47,E2 11933.47} C_VEL
LIN {X 0,Y 266.139,Z 1091.932,A -85,B 0,C 180,E1 11929.177,E2 11929.177} C_VEL
LIN {X 0,Y 276.246,Z 1080.2,A -85,B 0,C 180,E1 11924.516,E2 11924.516} C_VEL
LIN {X 0,Y 285.779,Z 1068.855,A -85,B 0,C 180,E1 11920.909,E2 11920.909} C_VEL
LIN {X 0,Y 297.477,Z 1054.385,A -85,B 0,C 180,E1 11917.192,E2 11917.192} C_VEL
LIN {X 0,Y 308.363,Z 1040.022,A -85,B 0,C 180,E1 11914.222,E2 11914.222} C_VEL
LIN {X 0,Y 320.324,Z 1023.24,A -85,B 0,C 180,E1 11911.38,E2 11911.38} C_VEL
LIN {X 0,Y 331.232,Z 1006.481,A -85,B 0,C 180,E1 11909.079,E2 11909.079} C_VEL
LIN {X 0,Y 342.257,Z 988.207,A -85,B 0,C 180,E1 11906.994,E2 11906.994} C_VEL
LIN {X 0,Y 352.867,Z 968.368,A -85,B 0,C 180,E1 11905.154,E2 11905.154} C_VEL
LIN {X 0,Y 361.999,Z 949.52,A -85,B 0,C 180,E1 11903.701,E2 11903.701} C_VEL
LIN {X 0,Y 371.35,Z 927.461,A -85,B 0,C 180,E1 11902.312,E2 11902.312} C_VEL
LIN {X 0,Y 378.354,Z 908.441,A -85,B 0,C 180,E1 11901.319,E2 11901.319} C_VEL
LIN {X 0,Y 385.762,Z 885.022,A -85,B 0,C 180,E1 11900.324,E2 11900.324} C_VEL
LIN {X 0,Y 391.504,Z 862.515,A -85,B 0,C 180,E1 11899.579,E2 11899.579} C_VEL
LIN {X 0,Y 396.363,Z 838.744,A -85,B 0,C 180,E1 11898.964,E2 11898.964} C_VEL
LIN {X 0,Y 399.743,Z 814.497,A -85,B 0,C 180,E1 11898.5,E2 11898.5} C_VEL
LIN {X 0,Y 415.465,Z 647.16,A -85,B 0,C 180,E1 11895.924,E2 11895.924} C_VEL
LIN {X 0,Y 412.711,Z 641.922,A -85,B 0,C 180,E1 11894.32,E2 11894.32} C_VEL
LIN {X 0,Y 411.116,Z 640.045,A -85,B 0,C 180,E1 11893.379,E2 11893.379} C_VEL
LIN {X 0,Y 408.34,Z 639.625,A -85,B 0,C 180,E1 11891.78,E2 11891.78} C_VEL
LIN {X 0,Y 405.866,Z 639.242,A -85,B 0,C 180,E1 11890.149,E2 11890.149} C_VEL
LIN {X 0,Y 405.045,Z 638.163,A -85,B 0,C 180,E1 11889.462,E2 11889.462} C_VEL
LIN {X 0,Y 402.193,Z 633.07,A -85,B 0,C 180,E1 11886.423,E2 11886.423} C_VEL
LIN {X 0,Y 400.064,Z 628.768,A -85,B 0,C 180,E1 11882.722,E2 11882.722} C_VEL
LIN {X 0,Y 399.208,Z 628.083,A -85,B 0,C 180,E1 11877.974,E2 11877.974} C_VEL
LIN {X 0,Y 400.235,Z 629.057,A -85,B 0,C 180,E1 11874.337,E2 11874.337} C_VEL
LIN {X 0,Y 402.757,Z 634.023,A -85,B 0,C 180,E1 11870.353,E2 11870.353} C_VEL
LIN {X 0,Y 405.315,Z 638.718,A -85,B 0,C 180,E1 11867.751,E2 11867.751} C_VEL
LIN {X 0,Y 407.653,Z 643.045,A -85,B 0,C 180,E1 11865.838,E2 11865.838} C_VEL
LIN {X 0,Y 411.931,Z 652.742,A -85,B 0,C 180,E1 11862.847,E2 11862.847} C_VEL
LIN {X 0,Y 412.57,Z 654.744,A -85,B 0,C 180,E1 11862.418,E2 11862.418} C_VEL
LIN {X 0,Y 395.947,Z 827.773,A -85,B 0,C 180,E1 11859.768,E2 11859.768} C_VEL
LIN {X 0,Y 391.69,Z 854.462,A -85,B 0,C 180,E1 11859.255,E2 11859.255} C_VEL
LIN {X 0,Y 386.862,Z 876.188,A -85,B 0,C 180,E1 11858.736,E2 11858.736} C_VEL
LIN {X 0,Y 379.733,Z 901.483,A -85,B 0,C 180,E1 11857.952,E2 11857.952} C_VEL
LIN {X 0,Y 372.746,Z 921.974,A -85,B 0,C 180,E1 11857.138,E2 11857.138} C_VEL
LIN {X 0,Y 363.478,Z 945.399,A -85,B 0,C 180,E1 11855.966,E2 11855.966} C_VEL
LIN {X 0,Y 354.403,Z 965.242,A -85,B 0,C 180,E1 11854.721,E2 11854.721} C_VEL
LIN {X 0,Y 343.997,Z 985.686,A -85,B 0,C 180,E1 11853.171,E2 11853.171} C_VEL
LIN {X 0,Y 332.771,Z 1005.159,A -85,B 0,C 180,E1 11851.329,E2 11851.329} C_VEL
LIN {X 0,Y 321.602,Z 1023.012,A -85,B 0,C 180,E1 11849.279,E2 11849.279} C_VEL
LIN {X 0,Y 309.525,Z 1040.581,A -85,B 0,C 180,E1 11846.791,E2 11846.791} C_VEL
LIN {X 0,Y 299.058,Z 1054.829,A -85,B 0,C 180,E1 11844.338,E2 11844.338} C_VEL
LIN {X 0,Y 286.818,Z 1070.586,A -85,B 0,C 180,E1 11841.025,E2 11841.025} C_VEL
LIN {X 0,Y 276.137,Z 1083.551,A -85,B 0,C 180,E1 11837.62,E2 11837.62} C_VEL
LIN {X 0,Y 265.549,Z 1096.172,A -85,B 0,C 180,E1 11833.556,E2 11833.556} C_VEL
LIN {X 0,Y 255.852,Z 1107.411,A -85,B 0,C 180,E1 11828.948,E2 11828.948} C_VEL
LIN {X 0,Y 248.223,Z 1116.489,A -85,B 0,C 180,E1 11824.329,E2 11824.329} C_VEL
LIN {X 0,Y 241.08,Z 1125.407,A -85,B 0,C 180,E1 11818.488,E2 11818.488} C_VEL
LIN {X 0,Y 236.792,Z 1131.417,A -85,B 0,C 180,E1 11813.386,E2 11813.386} C_VEL
LIN {X 0,Y 233.517,Z 1137.06,A -85,B 0,C 180,E1 11806.928,E2 11806.928} C_VEL
LIN {X 0,Y 232.312,Z 1140.165,A -85,B 0,C 180,E1 11801.671,E2 11801.671} C_VEL
LIN {X 0,Y 232.033,Z 1142.005,A -85,B 0,C 180,E1 11796.682,E2 11796.682} C_VEL
LIN {X 0,Y 232.091,Z 1142.74,A -85,B 0,C 180,E1 11791.728,E2 11791.728} C_VEL
LIN {X 0,Y 232.067,Z 1142.335,A -85,B 0,C 180,E1 11787.036,E2 11787.036} C_VEL
LIN {X 0,Y 232.045,Z 1140.716,A -85,B 0,C 180,E1 11782.074,E2 11782.074} C_VEL
LIN {X 0,Y 232.444,Z 1138.135,A -85,B 0,C 180,E1 11777.327,E2 11777.327} C_VEL
LIN {X 0,Y 233.731,Z 1134.3,A -85,B 0,C 180,E1 11772.318,E2 11772.318} C_VEL
LIN {X 0,Y 236.809,Z 1128.141,A -85,B 0,C 180,E1 11766.351,E2 11766.351} C_VEL
LIN {X 0,Y 241.354,Z 1120.73,A -85,B 0,C 180,E1 11760.944,E2 11760.944} C_VEL
LIN {X 0,Y 247.813,Z 1111.576,A -85,B 0,C 180,E1 11755.606,E2 11755.606} C_VEL
LIN {X 0,Y 255.75,Z 1100.778,A -85,B 0,C 180,E1 11750.701,E2 11750.701} C_VEL
LIN {X 0,Y 265.315,Z 1088.257,A -85,B 0,C 180,E1 11746.097,E2 11746.097} C_VEL
LIN {X 0,Y 275.297,Z 1074.829,A -85,B 0,C 180,E1 11742.188,E2 11742.188} C_VEL
LIN {X 0,Y 285.852,Z 1060.381,A -85,B 0,C 180,E1 11738.735,E2 11738.735} C_VEL
LIN {X 0,Y 297.332,Z 1043.674,A -85,B 0,C 180,E1 11735.529,E2 11735.529} C_VEL
LIN {X 0,Y 308.013,Z 1027.265,A -85,B 0,C 180,E1 11732.948,E2 11732.948} C_VEL
LIN {X 0,Y 319.627,Z 1007.861,A -85,B 0,C 180,E1 11730.475,E2 11730.475} C_VEL
LIN {X 0,Y 329.249,Z 990.346,A -85,B 0,C 180,E1 11728.638,E2 11728.638} C_VEL
LIN {X 0,Y 340.352,Z 967.994,A -85,B 0,C 180,E1 11726.735,E2 11726.735} C_VEL
LIN {X 0,Y 348.726,Z 949.014,A -85,B 0,C 180,E1 11725.419,E2 11725.419} C_VEL
LIN {X 0,Y 357.306,Z 927.146,A -85,B 0,C 180,E1 11724.176,E2 11724.176} C_VEL
LIN {X 0,Y 364.46,Z 905.672,A -85,B 0,C 180,E1 11723.209,E2 11723.209} C_VEL
LIN {X 0,Y 370.695,Z 883.855,A -85,B 0,C 180,E1 11722.42,E2 11722.42} C_VEL
LIN {X 0,Y 376.261,Z 859.263,A -85,B 0,C 180,E1 11721.742,E2 11721.742} C_VEL
LIN {X 0,Y 380.089,Z 836.749,A -85,B 0,C 180,E1 11721.251,E2 11721.251} C_VEL
LIN {X 0,Y 383.617,Z 803.475,A -85,B 0,C 180,E1 11720.68,E2 11720.68} C_VEL
LIN {X 0,Y 397.991,Z 643.737,A -85,B 0,C 180,E1 11718.152,E2 11718.152} C_VEL
LIN {X 0,Y 393.813,Z 634.247,A -85,B 0,C 180,E1 11715.839,E2 11715.839} C_VEL
LIN {X 0,Y 391.055,Z 628.424,A -85,B 0,C 180,E1 11714.134,E2 11714.134} C_VEL
LIN {X 0,Y 386.849,Z 621.008,A -85,B 0,C 180,E1 11711.178,E2 11711.178} C_VEL
LIN {X 0,Y 384.068,Z 616.334,A -85,B 0,C 180,E1 11708.76,E2 11708.76} C_VEL
LIN {X 0,Y 381.998,Z 612.651,A -85,B 0,C 180,E1 11706.463,E2 11706.463} C_VEL
LIN {X 0,Y 379.732,Z 608.274,A -85,B 0,C 180,E1 11702.641,E2 11702.641} C_VEL
LIN {X 0,Y 378.743,Z 607.514,A -85,B 0,C 180,E1 11697.428,E2 11697.428} C_VEL
LIN {X 0,Y 379.73,Z 608.363,A -85,B 0,C 180,E1 11693.802,E2 11693.802} C_VEL
LIN {X 0,Y 381.829,Z 612.468,A -85,B 0,C 180,E1 11690.2,E2 11690.2} C_VEL
LIN {X 0,Y 382.749,Z 614.104,A -85,B 0,C 180,E1 11689.082,E2 11689.082} C_VEL
LIN {X 0,Y 385.291,Z 618.418,A -85,B 0,C 180,E1 11686.569,E2 11686.569} C_VEL
LIN {X 0,Y 388.127,Z 623.349,A -85,B 0,C 180,E1 11684.306,E2 11684.306} C_VEL
LIN {X 0,Y 392.379,Z 630.924,A -85,B 0,C 180,E1 11681.503,E2 11681.503} C_VEL
LIN {X 0,Y 397.557,Z 640.561,A -85,B 0,C 180,E1 11678.65,E2 11678.65} C_VEL
LIN {X 0,Y 398.044,Z 641.811,A -85,B 0,C 180,E1 11678.388,E2 11678.388} C_VEL
LIN {X 0,Y 381.906,Z 817.966,A -85,B 0,C 180,E1 11675.597,E2 11675.597} C_VEL
LIN {X 0,Y 377.913,Z 844.425,A -85,B 0,C 180,E1 11675.03,E2 11675.03} C_VEL
LIN {X 0,Y 373.671,Z 865.025,A -85,B 0,C 180,E1 11674.44,E2 11674.44} C_VEL
LIN {X 0,Y 367.406,Z 889.304,A -85,B 0,C 180,E1 11673.556,E2 11673.556} C_VEL
LIN {X 0,Y 360.925,Z 909.822,A -85,B 0,C 180,E1 11672.611,E2 11672.611} C_VEL
LIN {X 0,Y 353.068,Z 931.474,A -85,B 0,C 180,E1 11671.393,E2 11671.393} C_VEL
LIN {X 0,Y 344.218,Z 952.236,A -85,B 0,C 180,E1 11669.956,E2 11669.956} C_VEL
LIN {X 0,Y 335.256,Z 971.129,A -85,B 0,C 180,E1 11668.375,E2 11668.375} C_VEL
LIN {X 0,Y 324.122,Z 992.031,A -85,B 0,C 180,E1 11666.242,E2 11666.242} C_VEL
LIN {X 0,Y 314.379,Z 1008.649,A -85,B 0,C 180,E1 11664.181,E2 11664.181} C_VEL
LIN {X 0,Y 302.15,Z 1027.763,A -85,B 0,C 180,E1 11661.285,E2 11661.285} C_VEL
LIN {X 0,Y 292.081,Z 1042.357,A -85,B 0,C 180,E1 11658.566,E2 11658.566} C_VEL
LIN {X 0,Y 280.4,Z 1058.341,A -85,B 0,C 180,E1 11654.915,E2 11654.915} C_VEL
LIN {X 0,Y 270.786,Z 1070.832,A -85,B 0,C 180,E1 11651.374,E2 11651.374} C_VEL
LIN {X 0,Y 260.897,Z 1083.415,A -85,B 0,C 180,E1 11646.992,E2 11646.992} C_VEL
LIN {X 0,Y 252.801,Z 1093.532,A -85,B 0,C 180,E1 11642.542,E2 11642.542} C_VEL
LIN {X 0,Y 245.486,Z 1103.014,A -85,B 0,C 180,E1 11637.384,E2 11637.384} C_VEL
LIN {X 0,Y 239.91,Z 1110.534,A -85,B 0,C 180,E1 11632.031,E2 11632.031} C_VEL
LIN {X 0,Y 236.134,Z 1116.375,A -85,B 0,C 180,E1 11626.735,E2 11626.735} C_VEL
LIN {X 0,Y 233.522,Z 1121.262,A -85,B 0,C 180,E1 11620.61,E2 11620.61} C_VEL
LIN {X 0,Y 232.51,Z 1123.945,A -85,B 0,C 180,E1 11615.676,E2 11615.676} C_VEL
LIN {X 0,Y 232.158,Z 1125.601,A -85,B 0,C 180,E1 11610.74,E2 11610.74} C_VEL
LIN {X 0,Y 232.107,Z 1126.263,A -85,B 0,C 180,E1 11605.553,E2 11605.553} C_VEL
LIN {X 0,Y 232.351,Z 1125.615,A -85,B 0,C 180,E1 11600.223,E2 11600.223} C_VEL
LIN {X 0,Y 233.091,Z 1124.015,A -85,B 0,C 180,E1 11595.339,E2 11595.339} C_VEL
LIN {X 0,Y 234.85,Z 1121.177,A -85,B 0,C 180,E1 11590.086,E2 11590.086} C_VEL
LIN {X 0,Y 238.623,Z 1116.121,A -85,B 0,C 180,E1 11583.898,E2 11583.898} C_VEL
LIN {X 0,Y 243.368,Z 1110.442,A -85,B 0,C 180,E1 11578.823,E2 11578.823} C_VEL
LIN {X 0,Y 250.655,Z 1102.292,A -85,B 0,C 180,E1 11573.247,E2 11573.247} C_VEL
LIN {X 0,Y 258.731,Z 1093.374,A -85,B 0,C 180,E1 11568.567,E2 11568.567} C_VEL
LIN {X 0,Y 268.529,Z 1082.633,A -85,B 0,C 180,E1 11564.056,E2 11564.056} C_VEL
LIN {X 0,Y 279.313,Z 1070.262,A -85,B 0,C 180,E1 11559.996,E2 11559.996} C_VEL
LIN {X 0,Y 290.744,Z 1056.783,A -85,B 0,C 180,E1 11556.414,E2 11556.414} C_VEL
LIN {X 0,Y 302.501,Z 1041.804,A -85,B 0,C 180,E1 11553.251,E2 11553.251} C_VEL
LIN {X 0,Y 313.724,Z 1026.667,A -85,B 0,C 180,E1 11550.623,E2 11550.623} C_VEL
LIN {X 0,Y 325.785,Z 1008.902,A -85,B 0,C 180,E1 11548.119,E2 11548.119} C_VEL
LIN {X 0,Y 336.018,Z 992.481,A -85,B 0,C 180,E1 11546.21,E2 11546.21} C_VEL
LIN {X 0,Y 347.823,Z 971.511,A -85,B 0,C 180,E1 11544.206,E2 11544.206} C_VEL
LIN {X 0,Y 356.84,Z 953.511,A -85,B 0,C 180,E1 11542.797,E2 11542.797} C_VEL
LIN {X 0,Y 366.289,Z 932.501,A -85,B 0,C 180,E1 11541.43,E2 11541.43} C_VEL
LIN {X 0,Y 374.63,Z 910.605,A -85,B 0,C 180,E1 11540.277,E2 11540.277} C_VEL
LIN {X 0,Y 381.978,Z 888.311,A -85,B 0,C 180,E1 11539.322,E2 11539.322} C_VEL
LIN {X 0,Y 388.301,Z 864.429,A -85,B 0,C 180,E1 11538.526,E2 11538.526} C_VEL
LIN {X 0,Y 392.839,Z 843.103,A -85,B 0,C 180,E1 11537.968,E2 11537.968} C_VEL
LIN {X 0,Y 396.783,Z 817.243,A -85,B 0,C 180,E1 11537.456,E2 11537.456} C_VEL
LIN {X 0,Y 412.618,Z 652.327,A -85,B 0,C 180,E1 11534.92,E2 11534.92} C_VEL
LIN {X 0,Y 408.476,Z 644.482,A -85,B 0,C 180,E1 11532.224,E2 11532.224} C_VEL
LIN {X 0,Y 405.257,Z 638.603,A -85,B 0,C 180,E1 11529.659,E2 11529.659} C_VEL
LIN {X 0,Y 405.045,Z 638.163,A -85,B 0,C 180,E1 11529.462,E2 11529.462} C_VEL
LIN {X 0,Y 404,Z 637.097,A -85,B 0,C 180,E1 11528.546,E2 11528.546} C_VEL
LIN {X 0,Y 402.226,Z 637.887,A -85,B 0,C 180,E1 11527.059,E2 11527.059} C_VEL
LIN {X 0,Y 400.378,Z 639.304,A -85,B 0,C 180,E1 11525.231,E2 11525.231} C_VEL
LIN {X 0,Y 399.834,Z 638.866,A -85,B 0,C 180,E1 11524.432,E2 11524.432} C_VEL
LIN {X 0,Y 399.025,Z 636.674,A -85,B 0,C 180,E1 11522.585,E2 11522.585} C_VEL
LIN {X 0,Y 398.246,Z 636.04,A -85,B 0,C 180,E1 11517.824,E2 11517.824} C_VEL
LIN {X 0,Y 399.193,Z 636.965,A -85,B 0,C 180,E1 11514.466,E2 11514.466} C_VEL
LIN {X 0,Y 401.592,Z 641.85,A -85,B 0,C 180,E1 11510.542,E2 11510.542} C_VEL
LIN {X 0,Y 404.012,Z 646.421,A -85,B 0,C 180,E1 11508.001,E2 11508.001} C_VEL
LIN {X 0,Y 406.197,Z 650.617,A -85,B 0,C 180,E1 11506.149,E2 11506.149} C_VEL
LIN {X 0,Y 409.923,Z 659.42,A -85,B 0,C 180,E1 11503.422,E2 11503.422} C_VEL
LIN {X 0,Y 393.429,Z 827.512,A -85,B 0,C 180,E1 11500.876,E2 11500.876} C_VEL
LIN {X 0,Y 389.12,Z 854.117,A -85,B 0,C 180,E1 11500.374,E2 11500.374} C_VEL
LIN {X 0,Y 384.194,Z 875.956,A -85,B 0,C 180,E1 11499.865,E2 11499.865} C_VEL
LIN {X 0,Y 377.216,Z 900.436,A -85,B 0,C 180,E1 11499.128,E2 11499.128} C_VEL
LIN {X 0,Y 370.114,Z 921.018,A -85,B 0,C 180,E1 11498.333,E2 11498.333} C_VEL
LIN {X 0,Y 361.089,Z 943.678,A -85,B 0,C 180,E1 11497.237,E2 11497.237} C_VEL
LIN {X 0,Y 351.427,Z 964.471,A -85,B 0,C 180,E1 11495.969,E2 11495.969} C_VEL
LIN {X 0,Y 340.855,Z 984.873,A -85,B 0,C 180,E1 11494.455,E2 11494.455} C_VEL
LIN {X 0,Y 329.317,Z 1004.506,A -85,B 0,C 180,E1 11492.637,E2 11492.637} C_VEL
LIN {X 0,Y 318.227,Z 1021.833,A -85,B 0,C 180,E1 11490.683,E2 11490.683} C_VEL
LIN {X 0,Y 305.11,Z 1040.477,A -85,B 0,C 180,E1 11488.08,E2 11488.08} C_VEL
LIN {X 0,Y 294.337,Z 1054.708,A -85,B 0,C 180,E1 11485.639,E2 11485.639} C_VEL
LIN {X 0,Y 281.7,Z 1070.433,A -85,B 0,C 180,E1 11482.33,E2 11482.33} C_VEL
LIN {X 0,Y 270.406,Z 1083.645,A -85,B 0,C 180,E1 11478.837,E2 11478.837} C_VEL
LIN {X 0,Y 259.112,Z 1096.541,A -85,B 0,C 180,E1 11474.614,E2 11474.614} C_VEL
LIN {X 0,Y 249.03,Z 1107.682,A -85,B 0,C 180,E1 11469.924,E2 11469.924} C_VEL
LIN {X 0,Y 240.395,Z 1117.511,A -85,B 0,C 180,E1 11464.739,E2 11464.739} C_VEL
LIN {X 0,Y 233.497,Z 1125.593,A -85,B 0,C 180,E1 11459.122,E2 11459.122} C_VEL
LIN {X 0,Y 228.723,Z 1131.96,A -85,B 0,C 180,E1 11453.442,E2 11453.442} C_VEL
LIN {X 0,Y 225.607,Z 1136.967,A -85,B 0,C 180,E1 11447.274,E2 11447.274} C_VEL
LIN {X 0,Y 224.364,Z 1139.898,A -85,B 0,C 180,E1 11442.091,E2 11442.091} C_VEL
LIN {X 0,Y 224.038,Z 1141.732,A -85,B 0,C 180,E1 11436.921,E2 11436.921} C_VEL
LIN {X 0,Y 224.093,Z 1142.459,A -85,B 0,C 180,E1 11431.79,E2 11431.79} C_VEL
LIN {X 0,Y 224.071,Z 1142.037,A -85,B 0,C 180,E1 11426.93,E2 11426.93} C_VEL
LIN {X 0,Y 224.057,Z 1140.407,A -85,B 0,C 180,E1 11421.79,E2 11421.79} C_VEL
LIN {X 0,Y 224.513,Z 1137.815,A -85,B 0,C 180,E1 11416.872,E2 11416.872} C_VEL
LIN {X 0,Y 225.936,Z 1133.968,A -85,B 0,C 180,E1 11411.687,E2 11411.687} C_VEL
LIN {X 0,Y 229.452,Z 1127.474,A -85,B 0,C 180,E1 11405.27,E2 11405.27} C_VEL
LIN {X 0,Y 234.086,Z 1120.449,A -85,B 0,C 180,E1 11400.016,E2 11400.016} C_VEL
LIN {X 0,Y 241,Z 1111.188,A -85,B 0,C 180,E1 11394.49,E2 11394.49} C_VEL
LIN {X 0,Y 249.363,Z 1100.378,A -85,B 0,C 180,E1 11389.489,E2 11389.489} C_VEL
LIN {X 0,Y 259.162,Z 1088.122,A -85,B 0,C 180,E1 11384.914,E2 11384.914} C_VEL
LIN {X 0,Y 269.78,Z 1074.39,A -85,B 0,C 180,E1 11380.879,E2 11380.879} C_VEL
LIN {X 0,Y 280.729,Z 1059.929,A -85,B 0,C 180,E1 11377.413,E2 11377.413} C_VEL
LIN {X 0,Y 292.596,Z 1043.191,A -85,B 0,C 180,E1 11374.209,E2 11374.209} C_VEL
LIN {X 0,Y 303.6,Z 1026.765,A -85,B 0,C 180,E1 11371.64,E2 11371.64} C_VEL
LIN {X 0,Y 315.269,Z 1007.771,A -85,B 0,C 180,E1 11369.237,E2 11369.237} C_VEL
LIN {X 0,Y 325.391,Z 989.781,A -85,B 0,C 180,E1 11367.368,E2 11367.368} C_VEL
LIN {X 0,Y 336.749,Z 967.372,A -85,B 0,C 180,E1 11365.491,E2 11365.491} C_VEL
LIN {X 0,Y 345.298,Z 948.358,A -85,B 0,C 180,E1 11364.194,E2 11364.194} C_VEL
LIN {X 0,Y 354.552,Z 924.947,A -85,B 0,C 180,E1 11362.904,E2 11362.904} C_VEL
LIN {X 0,Y 361.338,Z 904.863,A -85,B 0,C 180,E1 11362.026,E2 11362.026} C_VEL
LIN {X 0,Y 367.927,Z 882.105,A -85,B 0,C 180,E1 11361.227,E2 11361.227} C_VEL
LIN {X 0,Y 373.365,Z 857.996,A -85,B 0,C 180,E1 11360.585,E2 11360.585} C_VEL
LIN {X 0,Y 377.378,Z 834.414,A -85,B 0,C 180,E1 11360.083,E2 11360.083} C_VEL
LIN {X 0,Y 381.194,Z 797.36,A -85,B 0,C 180,E1 11359.467,E2 11359.467} C_VEL
LIN {X 0,Y 394.903,Z 648.354,A -85,B 0,C 180,E1 11357.128,E2 11357.128} C_VEL
LIN {X 0,Y 390.689,Z 638.478,A -85,B 0,C 180,E1 11354.601,E2 11354.601} C_VEL
LIN {X 0,Y 388.295,Z 633.851,A -85,B 0,C 180,E1 11353.022,E2 11353.022} C_VEL
LIN {X 0,Y 384.937,Z 627.852,A -85,B 0,C 180,E1 11350.476,E2 11350.476} C_VEL
LIN {X 0,Y 382.7,Z 623.908,A -85,B 0,C 180,E1 11348.413,E2 11348.413} C_VEL
LIN {X 0,Y 380.772,Z 620.393,A -85,B 0,C 180,E1 11346.181,E2 11346.181} C_VEL
LIN {X 0,Y 378.534,Z 615.973,A -85,B 0,C 180,E1 11342.119,E2 11342.119} C_VEL
LIN {X 0,Y 377.836,Z 615.528,A -85,B 0,C 180,E1 11336.814,E2 11336.814} C_VEL
LIN {X 0,Y 378.687,Z 616.278,A -85,B 0,C 180,E1 11333.937,E2 11333.937} C_VEL
LIN {X 0,Y 380.858,Z 620.485,A -85,B 0,C 180,E1 11330.174,E2 11330.174} C_VEL
LIN {X 0,Y 383.97,Z 626.127,A -85,B 0,C 180,E1 11326.829,E2 11326.829} C_VEL
LIN {X 0,Y 386.736,Z 631.077,A -85,B 0,C 180,E1 11324.556,E2 11324.556} C_VEL
LIN {X 0,Y 391.134,Z 639.146,A -85,B 0,C 180,E1 11321.596,E2 11321.596} C_VEL
LIN {X 0,Y 394.95,Z 646.641,A -85,B 0,C 180,E1 11319.407,E2 11319.407} C_VEL
LIN {X 0,Y 378.865,Z 818.363,A -85,B 0,C 180,E1 11316.711,E2 11316.711} C_VEL
LIN {X 0,Y 374.824,Z 844.644,A -85,B 0,C 180,E1 11316.154,E2 11316.154} C_VEL
LIN {X 0,Y 370.502,Z 865.262,A -85,B 0,C 180,E1 11315.574,E2 11315.574} C_VEL
LIN {X 0,Y 364.326,Z 888.887,A -85,B 0,C 180,E1 11314.731,E2 11314.731} C_VEL
LIN {X 0,Y 357.331,Z 910.606,A -85,B 0,C 180,E1 11313.745,E2 11313.745} C_VEL
LIN {X 0,Y 348.939,Z 933.121,A -85,B 0,C 180,E1 11312.484,E2 11312.484} C_VEL
LIN {X 0,Y 339.777,Z 953.973,A -85,B 0,C 180,E1 11311.038,E2 11311.038} C_VEL
LIN {X 0,Y 329.685,Z 974.627,A -85,B 0,C 180,E1 11309.297,E2 11309.297} C_VEL
LIN {X 0,Y 318.677,Z 994.385,A -85,B 0,C 180,E1 11307.234,E2 11307.234} C_VEL
LIN {X 0,Y 307.429,Z 1012.939,A -85,B 0,C 180,E1 11304.884,E2 11304.884} C_VEL
LIN {X 0,Y 296.037,Z 1029.876,A -85,B 0,C 180,E1 11302.219,E2 11302.219} C_VEL
LIN {X 0,Y 284.992,Z 1045.349,A -85,B 0,C 180,E1 11299.263,E2 11299.263} C_VEL
LIN {X 0,Y 273.576,Z 1060.225,A -85,B 0,C 180,E1 11295.726,E2 11295.726} C_VEL
LIN {X 0,Y 263.763,Z 1072.506,A -85,B 0,C 180,E1 11292.143,E2 11292.143} C_VEL
LIN {X 0,Y 253.108,Z 1085.393,A -85,B 0,C 180,E1 11287.435,E2 11287.435} C_VEL
LIN {X 0,Y 245.262,Z 1094.819,A -85,B 0,C 180,E1 11283.113,E2 11283.113} C_VEL
LIN {X 0,Y 237.18,Z 1104.736,A -85,B 0,C 180,E1 11277.356,E2 11277.356} C_VEL
LIN {X 0,Y 231.997,Z 1111.479,A -85,B 0,C 180,E1 11272.289,E2 11272.289} C_VEL
LIN {X 0,Y 227.853,Z 1117.655,A -85,B 0,C 180,E1 11266.311,E2 11266.311} C_VEL
LIN {X 0,Y 225.471,Z 1121.892,A -85,B 0,C 180,E1 11260.476,E2 11260.476} C_VEL
LIN {X 0,Y 224.475,Z 1124.476,A -85,B 0,C 180,E1 11255.367,E2 11255.367} C_VEL
LIN {X 0,Y 224.143,Z 1126.163,A -85,B 0,C 180,E1 11249.744,E2 11249.744} C_VEL
LIN {X 0,Y 224.138,Z 1126.464,A -85,B 0,C 180,E1 11244.368,E2 11244.368} C_VEL
LIN {X 0,Y 224.393,Z 1125.853,A -85,B 0,C 180,E1 11239.733,E2 11239.733} C_VEL
LIN {X 0,Y 225.212,Z 1124.279,A -85,B 0,C 180,E1 11234.814,E2 11234.814} C_VEL
LIN {X 0,Y 227.274,Z 1121.278,A -85,B 0,C 180,E1 11229.123,E2 11229.123} C_VEL
LIN {X 0,Y 231.436,Z 1116.108,A -85,B 0,C 180,E1 11222.744,E2 11222.744} C_VEL
LIN {X 0,Y 236.583,Z 1110.37,A -85,B 0,C 180,E1 11217.537,E2 11217.537} C_VEL
LIN {X 0,Y 244.767,Z 1101.696,A -85,B 0,C 180,E1 11211.616,E2 11211.616} C_VEL
LIN {X 0,Y 253.327,Z 1092.762,A -85,B 0,C 180,E1 11206.934,E2 11206.934} C_VEL
LIN {X 0,Y 264.848,Z 1080.525,A -85,B 0,C 180,E1 11201.949,E2 11201.949} C_VEL
LIN {X 0,Y 275.19,Z 1069.151,A -85,B 0,C 180,E1 11198.295,E2 11198.295} C_VEL
LIN {X 0,Y 288.377,Z 1053.851,A -85,B 0,C 180,E1 11194.389,E2 11194.389} C_VEL
LIN {X 0,Y 299.37,Z 1040.22,A -85,B 0,C 180,E1 11191.603,E2 11191.603} C_VEL
LIN {X 0,Y 312.396,Z 1022.856,A -85,B 0,C 180,E1 11188.717,E2 11188.717} C_VEL
LIN {X 0,Y 323.537,Z 1006.586,A -85,B 0,C 180,E1 11186.534,E2 11186.534} C_VEL
LIN {X 0,Y 335.126,Z 988.217,A -85,B 0,C 180,E1 11184.493,E2 11184.493} C_VEL
LIN {X 0,Y 345.887,Z 968.928,A -85,B 0,C 180,E1 11182.754,E2 11182.754} C_VEL
LIN {X 0,Y 355.358,Z 950.18,A -85,B 0,C 180,E1 11181.352,E2 11181.352} C_VEL
LIN {X 0,Y 365.297,Z 927.597,A -85,B 0,C 180,E1 11179.977,E2 11179.977} C_VEL
LIN {X 0,Y 372.759,Z 908.004,A -85,B 0,C 180,E1 11178.994,E2 11178.994} C_VEL
LIN {X 0,Y 380.818,Z 882.883,A -85,B 0,C 180,E1 11177.984,E2 11177.984} C_VEL
LIN {X 0,Y 386.412,Z 861.387,A -85,B 0,C 180,E1 11177.31,E2 11177.31} C_VEL
LIN {X 0,Y 391.615,Z 835.589,A -85,B 0,C 180,E1 11176.69,E2 11176.69} C_VEL
LIN {X 0,Y 394.748,Z 813.246,A -85,B 0,C 180,E1 11176.287,E2 11176.287} C_VEL
LIN {X 0,Y 409.934,Z 657.767,A -85,B 0,C 180,E1 11173.938,E2 11173.938} C_VEL
LIN {X 0,Y 406.081,Z 650.332,A -85,B 0,C 180,E1 11171.217,E2 11171.217} C_VEL
LIN {X 0,Y 403,Z 644.573,A -85,B 0,C 180,E1 11168.489,E2 11168.489} C_VEL
LIN {X 0,Y 400.984,Z 640.806,A -85,B 0,C 180,E1 11166.155,E2 11166.155} C_VEL
LIN {X 0,Y 399.834,Z 638.866,A -85,B 0,C 180,E1 11164.432,E2 11164.432} C_VEL
LIN {X 0,Y 399.211,Z 638.627,A -85,B 0,C 180,E1 11163.405,E2 11163.405} C_VEL
LIN {X 0,Y 398.196,Z 640.821,A -85,B 0,C 180,E1 11161.833,E2 11161.833} C_VEL
LIN {X 0,Y 397.353,Z 643.71,A -85,B 0,C 180,E1 11160.006,E2 11160.006} C_VEL
LIN {X 0,Y 397.243,Z 643.99,A -85,B 0,C 180,E1 11159.357,E2 11159.357} C_VEL
LIN {X 0,Y 398.106,Z 644.666,A -85,B 0,C 180,E1 11154.74,E2 11154.74} C_VEL
LIN {X 0,Y 400.432,Z 649.675,A -85,B 0,C 180,E1 11150.732,E2 11150.732} C_VEL
LIN {X 0,Y 402.717,Z 654.123,A -85,B 0,C 180,E1 11148.253,E2 11148.253} C_VEL
LIN {X 0,Y 404.754,Z 658.188,A -85,B 0,C 180,E1 11146.463,E2 11146.463} C_VEL
LIN {X 0,Y 407.343,Z 664.728,A -85,B 0,C 180,E1 11144.43,E2 11144.43} C_VEL
LIN {X 0,Y 391.074,Z 827.141,A -85,B 0,C 180,E1 11142,E2 11142} C_VEL
LIN {X 0,Y 386.69,Z 853.814,A -85,B 0,C 180,E1 11141.507,E2 11141.507} C_VEL
LIN {X 0,Y 381.703,Z 875.615,A -85,B 0,C 180,E1 11141.011,E2 11141.011} C_VEL
LIN {X 0,Y 374.435,Z 900.67,A -85,B 0,C 180,E1 11140.274,E2 11140.274} C_VEL
LIN {X 0,Y 367.225,Z 921.189,A -85,B 0,C 180,E1 11139.498,E2 11139.498} C_VEL
LIN {X 0,Y 358.05,Z 943.756,A -85,B 0,C 180,E1 11138.426,E2 11138.426} C_VEL
LIN {X 0,Y 348.214,Z 964.513,A -85,B 0,C 180,E1 11137.183,E2 11137.183} C_VEL
LIN {X 0,Y 337.135,Z 985.41,A -85,B 0,C 180,E1 11135.653,E2 11135.653} C_VEL
LIN {X 0,Y 325.654,Z 1004.463,A -85,B 0,C 180,E1 11133.909,E2 11133.909} C_VEL
LIN {X 0,Y 314.306,Z 1021.767,A -85,B 0,C 180,E1 11131.983,E2 11131.983} C_VEL
LIN {X 0,Y 301.176,Z 1039.95,A -85,B 0,C 180,E1 11129.472,E2 11129.472} C_VEL
LIN {X 0,Y 289.578,Z 1054.833,A -85,B 0,C 180,E1 11126.937,E2 11126.937} C_VEL
LIN {X 0,Y 275.48,Z 1071.695,A -85,B 0,C 180,E1 11123.336,E2 11123.336} C_VEL
LIN {X 0,Y 264.12,Z 1084.502,A -85,B 0,C 180,E1 11119.883,E2 11119.883} C_VEL
LIN {X 0,Y 251.252,Z 1098.439,A -85,B 0,C 180,E1 11115.103,E2 11115.103} C_VEL
LIN {X 0,Y 241.927,Z 1108.336,A -85,B 0,C 180,E1 11110.77,E2 11110.77} C_VEL
LIN {X 0,Y 232.23,Z 1118.745,A -85,B 0,C 180,E1 11104.935,E2 11104.935} C_VEL
LIN {X 0,Y 225.865,Z 1125.872,A -85,B 0,C 180,E1 11099.724,E2 11099.724} C_VEL
LIN {X 0,Y 220.654,Z 1132.461,A -85,B 0,C 180,E1 11093.502,E2 11093.502} C_VEL
LIN {X 0,Y 217.61,Z 1137.041,A -85,B 0,C 180,E1 11087.378,E2 11087.378} C_VEL
LIN {X 0,Y 216.348,Z 1139.871,A -85,B 0,C 180,E1 11082.004,E2 11082.004} C_VEL
LIN {X 0,Y 216.032,Z 1141.747,A -85,B 0,C 180,E1 11076.111,E2 11076.111} C_VEL
LIN {X 0,Y 216.106,Z 1142.141,A -85,B 0,C 180,E1 11070.795,E2 11070.795} C_VEL
LIN {X 0,Y 216.072,Z 1141.529,A -85,B 0,C 180,E1 11066.02,E2 11066.02} C_VEL
LIN {X 0,Y 216.086,Z 1139.979,A -85,B 0,C 180,E1 11061.216,E2 11061.216} C_VEL
LIN {X 0,Y 216.647,Z 1137.327,A -85,B 0,C 180,E1 11056.114,E2 11056.114} C_VEL
LIN {X 0,Y 218.392,Z 1133.205,A -85,B 0,C 180,E1 11050.475,E2 11050.475} C_VEL
LIN {X 0,Y 222.368,Z 1126.491,A -85,B 0,C 180,E1 11043.854,E2 11043.854} C_VEL
LIN {X 0,Y 227.497,Z 1119.354,A -85,B 0,C 180,E1 11038.464,E2 11038.464} C_VEL
LIN {X 0,Y 235.754,Z 1108.912,A -85,B 0,C 180,E1 11032.357,E2 11032.357} C_VEL
LIN {X 0,Y 243.98,Z 1098.92,A -85,B 0,C 180,E1 11027.769,E2 11027.769} C_VEL
LIN {X 0,Y 255.126,Z 1085.456,A -85,B 0,C 180,E1 11022.87,E2 11022.87} C_VEL
LIN {X 0,Y 264.982,Z 1073.235,A -85,B 0,C 180,E1 11019.326,E2 11019.326} C_VEL
LIN {X 0,Y 277.01,Z 1057.815,A -85,B 0,C 180,E1 11015.692,E2 11015.692} C_VEL
LIN {X 0,Y 288.694,Z 1041.764,A -85,B 0,C 180,E1 11012.687,E2 11012.687} C_VEL
LIN {X 0,Y 300.767,Z 1024.177,A -85,B 0,C 180,E1 11010.001,E2 11010.001} C_VEL
LIN {X 0,Y 312.158,Z 1005.842,A -85,B 0,C 180,E1 11007.761,E2 11007.761} C_VEL
LIN {X 0,Y 323.232,Z 986.506,A -85,B 0,C 180,E1 11005.817,E2 11005.817} C_VEL
LIN {X 0,Y 333.702,Z 965.928,A -85,B 0,C 180,E1 11004.161,E2 11004.161} C_VEL
LIN {X 0,Y 342.835,Z 945.877,A -85,B 0,C 180,E1 11002.834,E2 11002.834} C_VEL
LIN {X 0,Y 352.168,Z 922.212,A -85,B 0,C 180,E1 11001.587,E2 11001.587} C_VEL
LIN {X 0,Y 359.204,Z 901.452,A -85,B 0,C 180,E1 11000.723,E2 11000.723} C_VEL
LIN {X 0,Y 366.357,Z 875.862,A -85,B 0,C 180,E1 10999.893,E2 10999.893} C_VEL
LIN {X 0,Y 371.131,Z 854.183,A -85,B 0,C 180,E1 10999.353,E2 10999.353} C_VEL
LIN {X 0,Y 375.392,Z 826.972,A -85,B 0,C 180,E1 10998.813,E2 10998.813} C_VEL
LIN {X 0,Y 391.948,Z 652.954,A -85,B 0,C 180,E1 10996.089,E2 10996.089} C_VEL
LIN {X 0,Y 387.916,Z 643.502,A -85,B 0,C 180,E1 10993.49,E2 10993.49} C_VEL
LIN {X 0,Y 383.94,Z 636.096,A -85,B 0,C 180,E1 10990.504,E2 10990.504} C_VEL
LIN {X 0,Y 381.418,Z 631.593,A -85,B 0,C 180,E1 10988.138,E2 10988.138} C_VEL
LIN {X 0,Y 379.555,Z 628.131,A -85,B 0,C 180,E1 10985.897,E2 10985.897} C_VEL
LIN {X 0,Y 377.497,Z 623.883,A -85,B 0,C 180,E1 10981.973,E2 10981.973} C_VEL
LIN {X 0,Y 376.862,Z 623.47,A -85,B 0,C 180,E1 10976.806,E2 10976.806} C_VEL
LIN {X 0,Y 377.647,Z 624.192,A -85,B 0,C 180,E1 10974.073,E2 10974.073} C_VEL
LIN {X 0,Y 380.102,Z 629.096,A -85,B 0,C 180,E1 10969.849,E2 10969.849} C_VEL
LIN {X 0,Y 382.714,Z 633.943,A -85,B 0,C 180,E1 10967.038,E2 10967.038} C_VEL
LIN {X 0,Y 385.449,Z 638.975,A -85,B 0,C 180,E1 10964.734,E2 10964.734} C_VEL
LIN {X 0,Y 389.774,Z 647.158,A -85,B 0,C 180,E1 10961.762,E2 10961.762} C_VEL
LIN {X 0,Y 391.945,Z 651.858,A -85,B 0,C 180,E1 10960.437,E2 10960.437} C_VEL
LIN {X 0,Y 375.979,Z 818.665,A -85,B 0,C 180,E1 10957.843,E2 10957.843} C_VEL
LIN {X 0,Y 371.848,Z 845.021,A -85,B 0,C 180,E1 10957.293,E2 10957.293} C_VEL
LIN {X 0,Y 367.44,Z 865.663,A -85,B 0,C 180,E1 10956.721,E2 10956.721} C_VEL
LIN {X 0,Y 361.002,Z 889.736,A -85,B 0,C 180,E1 10955.873,E2 10955.873} C_VEL
LIN {X 0,Y 354.207,Z 910.456,A -85,B 0,C 180,E1 10954.948,E2 10954.948} C_VEL
LIN {X 0,Y 345.713,Z 932.91,A -85,B 0,C 180,E1 10953.715,E2 10953.715} C_VEL
LIN {X 0,Y 336.497,Z 953.525,A -85,B 0,C 180,E1 10952.313,E2 10952.313} C_VEL
LIN {X 0,Y 327.14,Z 972.352,A -85,B 0,C 180,E1 10950.765,E2 10950.765} C_VEL
LIN {X 0,Y 315.658,Z 992.848,A -85,B 0,C 180,E1 10948.702,E2 10948.702} C_VEL
LIN {X 0,Y 305.624,Z 1009.116,A -85,B 0,C 180,E1 10946.711,E2 10946.711} C_VEL
LIN {X 0,Y 293.133,Z 1027.645,A -85,B 0,C 180,E1 10943.942,E2 10943.942} C_VEL
LIN {X 0,Y 282.264,Z 1042.485,A -85,B 0,C 180,E1 10941.199,E2 10941.199} C_VEL
LIN {X 0,Y 270.036,Z 1058.189,A -85,B 0,C 180,E1 10937.63,E2 10937.63} C_VEL
LIN {X 0,Y 259.351,Z 1071.076,A -85,B 0,C 180,E1 10933.945,E2 10933.945} C_VEL
LIN {X 0,Y 248.583,Z 1083.725,A -85,B 0,C 180,E1 10929.46,E2 10929.46} C_VEL
LIN {X 0,Y 239.271,Z 1094.319,A -85,B 0,C 180,E1 10924.634,E2 10924.634} C_VEL
LIN {X 0,Y 231.223,Z 1103.734,A -85,B 0,C 180,E1 10919.252,E2 10919.252} C_VEL
LIN {X 0,Y 224.977,Z 1111.249,A -85,B 0,C 180,E1 10913.578,E2 10913.578} C_VEL
LIN {X 0,Y 220.56,Z 1117.312,A -85,B 0,C 180,E1 10907.682,E2 10907.682} C_VEL
LIN {X 0,Y 217.738,Z 1121.906,A -85,B 0,C 180,E1 10901.389,E2 10901.389} C_VEL
LIN {X 0,Y 216.573,Z 1124.567,A -85,B 0,C 180,E1 10896.096,E2 10896.096} C_VEL
LIN {X 0,Y 216.17,Z 1126.201,A -85,B 0,C 180,E1 10890.795,E2 10890.795} C_VEL
LIN {X 0,Y 216.121,Z 1126.828,A -85,B 0,C 180,E1 10885.223,E2 10885.223} C_VEL
LIN {X 0,Y 216.409,Z 1126.189,A -85,B 0,C 180,E1 10879.619,E2 10879.619} C_VEL
LIN {X 0,Y 217.349,Z 1124.543,A -85,B 0,C 180,E1 10874.251,E2 10874.251} C_VEL
LIN {X 0,Y 219.615,Z 1121.534,A -85,B 0,C 180,E1 10868.359,E2 10868.359} C_VEL
LIN {X 0,Y 223.891,Z 1116.591,A -85,B 0,C 180,E1 10862.035,E2 10862.035} C_VEL
LIN {X 0,Y 229.322,Z 1110.891,A -85,B 0,C 180,E1 10856.675,E2 10856.675} C_VEL
LIN {X 0,Y 237.914,Z 1102.297,A -85,B 0,C 180,E1 10850.608,E2 10850.608} C_VEL
LIN {X 0,Y 246.388,Z 1093.857,A -85,B 0,C 180,E1 10846.056,E2 10846.056} C_VEL
LIN {X 0,Y 257.393,Z 1082.789,A -85,B 0,C 180,E1 10841.33,E2 10841.33} C_VEL
LIN {X 0,Y 268.827,Z 1070.679,A -85,B 0,C 180,E1 10837.321,E2 10837.321} C_VEL
LIN {X 0,Y 281.269,Z 1056.974,A -85,B 0,C 180,E1 10833.681,E2 10833.681} C_VEL
LIN {X 0,Y 293.754,Z 1042.005,A -85,B 0,C 180,E1 10830.551,E2 10830.551} C_VEL
LIN {X 0,Y 306.365,Z 1025.908,A -85,B 0,C 180,E1 10827.813,E2 10827.813} C_VEL
LIN {X 0,Y 318.833,Z 1008.276,A -85,B 0,C 180,E1 10825.418,E2 10825.418} C_VEL
LIN {X 0,Y 330.259,Z 990.687,A -85,B 0,C 180,E1 10823.456,E2 10823.456} C_VEL
LIN {X 0,Y 342.013,Z 970.361,A -85,B 0,C 180,E1 10821.613,E2 10821.613} C_VEL
LIN {X 0,Y 351.25,Z 952.547,A -85,B 0,C 180,E1 10820.285,E2 10820.285} C_VEL
LIN {X 0,Y 361.483,Z 930.165,A -85,B 0,C 180,E1 10818.914,E2 10818.914} C_VEL
LIN {X 0,Y 369.18,Z 910.539,A -85,B 0,C 180,E1 10817.929,E2 10817.929} C_VEL
LIN {X 0,Y 376.965,Z 887.568,A -85,B 0,C 180,E1 10816.99,E2 10816.99} C_VEL
LIN {X 0,Y 383.346,Z 863.925,A -85,B 0,C 180,E1 10816.243,E2 10816.243} C_VEL
LIN {X 0,Y 388.449,Z 840.365,A -85,B 0,C 180,E1 10815.663,E2 10815.663} C_VEL
LIN {X 0,Y 392.086,Z 815.873,A -85,B 0,C 180,E1 10815.213,E2 10815.213} C_VEL
LIN {X 0,Y 407.319,Z 663.138,A -85,B 0,C 180,E1 10812.908,E2 10812.908} C_VEL
LIN {X 0,Y 403.649,Z 655.891,A -85,B 0,C 180,E1 10810.058,E2 10810.058} C_VEL
LIN {X 0,Y 401.592,Z 652.041,A -85,B 0,C 180,E1 10808.087,E2 10808.087} C_VEL
LIN {X 0,Y 399.893,Z 648.682,A -85,B 0,C 180,E1 10806.028,E2 10806.028} C_VEL
LIN {X 0,Y 397.989,Z 644.579,A -85,B 0,C 180,E1 10802.448,E2 10802.448} C_VEL
LIN {X 0,Y 397.243,Z 643.99,A -85,B 0,C 180,E1 10799.357,E2 10799.357} C_VEL
LIN {X 0,Y 397.119,Z 644.962,A -85,B 0,C 180,E1 10798.167,E2 10798.167} C_VEL
LIN {X 0,Y 396.944,Z 649.286,A -85,B 0,C 180,E1 10796.248,E2 10796.248} C_VEL
LIN {X 0,Y 397.177,Z 653.008,A -85,B 0,C 180,E1 10794.544,E2 10794.544} C_VEL
LIN {X 0,Y 397.231,Z 653.236,A -85,B 0,C 180,E1 10794.385,E2 10794.385} C_VEL
LIN {X 0,Y 399.224,Z 657.368,A -85,B 0,C 180,E1 10790.994,E2 10790.994} C_VEL
LIN {X 0,Y 401.429,Z 661.825,A -85,B 0,C 180,E1 10788.506,E2 10788.506} C_VEL
LIN {X 0,Y 403.323,Z 665.758,A -85,B 0,C 180,E1 10786.779,E2 10786.779} C_VEL
LIN {X 0,Y 404.881,Z 670.108,A -85,B 0,C 180,E1 10785.45,E2 10785.45} C_VEL
LIN {X 0,Y 388.845,Z 827.006,A -85,B 0,C 180,E1 10783.133,E2 10783.133} C_VEL
LIN {X 0,Y 384.403,Z 853.573,A -85,B 0,C 180,E1 10782.651,E2 10782.651} C_VEL
LIN {X 0,Y 379.324,Z 875.456,A -85,B 0,C 180,E1 10782.168,E2 10782.168} C_VEL
LIN {X 0,Y 371.807,Z 900.907,A -85,B 0,C 180,E1 10781.437,E2 10781.437} C_VEL
LIN {X 0,Y 364.49,Z 921.361,A -85,B 0,C 180,E1 10780.68,E2 10780.68} C_VEL
LIN {X 0,Y 354.743,Z 944.734,A -85,B 0,C 180,E1 10779.586,E2 10779.586} C_VEL
LIN {X 0,Y 345.574,Z 963.744,A -85,B 0,C 180,E1 10778.472,E2 10778.472} C_VEL
LIN {X 0,Y 334.989,Z 983.425,A -85,B 0,C 180,E1 10777.077,E2 10777.077} C_VEL
LIN {X 0,Y 322.941,Z 1003.203,A -85,B 0,C 180,E1 10775.332,E2 10775.332} C_VEL
LIN {X 0,Y 311.691,Z 1020.034,A -85,B 0,C 180,E1 10773.512,E2 10773.512} C_VEL
LIN {X 0,Y 297.49,Z 1039.339,A -85,B 0,C 180,E1 10770.914,E2 10770.914} C_VEL
LIN {X 0,Y 285.371,Z 1054.466,A -85,B 0,C 180,E1 10768.368,E2 10768.368} C_VEL
LIN {X 0,Y 271.198,Z 1070.927,A -85,B 0,C 180,E1 10764.889,E2 10764.889} C_VEL
LIN {X 0,Y 259.464,Z 1083.696,A -85,B 0,C 180,E1 10761.472,E2 10761.472} C_VEL
LIN {X 0,Y 247.052,Z 1096.682,A -85,B 0,C 180,E1 10757.102,E2 10757.102} C_VEL
LIN {X 0,Y 236.62,Z 1107.2,A -85,B 0,C 180,E1 10752.541,E2 10752.541} C_VEL
LIN {X 0,Y 226.944,Z 1117.095,A -85,B 0,C 180,E1 10747.111,E2 10747.111} C_VEL
LIN {X 0,Y 219.295,Z 1125.017,A -85,B 0,C 180,E1 10741.318,E2 10741.318} C_VEL
LIN {X 0,Y 213.704,Z 1131.475,A -85,B 0,C 180,E1 10735.2,E2 10735.2} C_VEL
LIN {X 0,Y 210.028,Z 1136.447,A -85,B 0,C 180,E1 10728.601,E2 10728.601} C_VEL
LIN {X 0,Y 208.491,Z 1139.364,A -85,B 0,C 180,E1 10723.027,E2 10723.027} C_VEL
LIN {X 0,Y 208.029,Z 1141.184,A -85,B 0,C 180,E1 10717.457,E2 10717.457} C_VEL
LIN {X 0,Y 208.097,Z 1141.899,A -85,B 0,C 180,E1 10711.927,E2 10711.927} C_VEL
LIN {X 0,Y 208.08,Z 1141.51,A -85,B 0,C 180,E1 10706.97,E2 10706.97} C_VEL
LIN {X 0,Y 208.078,Z 1139.906,A -85,B 0,C 180,E1 10701.433,E2 10701.433} C_VEL
LIN {X 0,Y 208.688,Z 1137.172,A -85,B 0,C 180,E1 10695.856,E2 10695.856} C_VEL
LIN {X 0,Y 210.544,Z 1133.087,A -85,B 0,C 180,E1 10690.005,E2 10690.005} C_VEL
LIN {X 0,Y 214.758,Z 1126.45,A -85,B 0,C 180,E1 10683.152,E2 10683.152} C_VEL
LIN {X 0,Y 220.164,Z 1119.351,A -85,B 0,C 180,E1 10677.594,E2 10677.594} C_VEL
LIN {X 0,Y 228.436,Z 1109.467,A -85,B 0,C 180,E1 10671.57,E2 10671.57} C_VEL
LIN {X 0,Y 236.95,Z 1099.576,A -85,B 0,C 180,E1 10666.873,E2 10666.873} C_VEL
LIN {X 0,Y 247.399,Z 1087.623,A -85,B 0,C 180,E1 10662.301,E2 10662.301} C_VEL
LIN {X 0,Y 259.089,Z 1073.643,A -85,B 0,C 180,E1 10658.133,E2 10658.133} C_VEL
LIN {X 0,Y 270.962,Z 1059.023,A -85,B 0,C 180,E1 10654.623,E2 10654.623} C_VEL
LIN {X 0,Y 283.541,Z 1042.331,A -85,B 0,C 180,E1 10651.461,E2 10651.461} C_VEL
LIN {X 0,Y 295.639,Z 1025.247,A -85,B 0,C 180,E1 10648.839,E2 10648.839} C_VEL
LIN {X 0,Y 307.86,Z 1006.203,A -85,B 0,C 180,E1 10646.507,E2 10646.507} C_VEL
LIN {X 0,Y 318.656,Z 987.826,A -85,B 0,C 180,E1 10644.666,E2 10644.666} C_VEL
LIN {X 0,Y 330.038,Z 966.127,A -85,B 0,C 180,E1 10642.926,E2 10642.926} C_VEL
LIN {X 0,Y 338.932,Z 947.04,A -85,B 0,C 180,E1 10641.675,E2 10641.675} C_VEL
LIN {X 0,Y 348.84,Z 922.602,A -85,B 0,C 180,E1 10640.398,E2 10640.398} C_VEL
LIN {X 0,Y 355.99,Z 901.934,A -85,B 0,C 180,E1 10639.551,E2 10639.551} C_VEL
LIN {X 0,Y 363.175,Z 876.945,A -85,B 0,C 180,E1 10638.75,E2 10638.75} C_VEL
LIN {X 0,Y 368.119,Z 855.055,A -85,B 0,C 180,E1 10638.21,E2 10638.21} C_VEL
LIN {X 0,Y 372.333,Z 829.716,A -85,B 0,C 180,E1 10637.705,E2 10637.705} C_VEL
LIN {X 0,Y 378.988,Z 762.767,A -85,B 0,C 180,E1 10636.648,E2 10636.648} C_VEL
LIN {X 0,Y 389.11,Z 657.765,A -85,B 0,C 180,E1 10635.043,E2 10635.043} C_VEL
LIN {X 0,Y 386.049,Z 650.482,A -85,B 0,C 180,E1 10632.946,E2 10632.946} C_VEL
LIN {X 0,Y 382.42,Z 643.5,A -85,B 0,C 180,E1 10630.089,E2 10630.089} C_VEL
LIN {X 0,Y 380.145,Z 639.277,A -85,B 0,C 180,E1 10627.861,E2 10627.861} C_VEL
LIN {X 0,Y 378.461,Z 636.005,A -85,B 0,C 180,E1 10625.762,E2 10625.762} C_VEL
LIN {X 0,Y 376.462,Z 631.792,A -85,B 0,C 180,E1 10621.826,E2 10621.826} C_VEL
LIN {X 0,Y 375.888,Z 631.413,A -85,B 0,C 180,E1 10616.798,E2 10616.798} C_VEL
LIN {X 0,Y 376.631,Z 632.206,A -85,B 0,C 180,E1 10614.133,E2 10614.133} C_VEL
LIN {X 0,Y 378.939,Z 636.926,A -85,B 0,C 180,E1 10610.047,E2 10610.047} C_VEL
LIN {X 0,Y 381.354,Z 641.54,A -85,B 0,C 180,E1 10607.354,E2 10607.354} C_VEL
LIN {X 0,Y 384.261,Z 647.035,A -85,B 0,C 180,E1 10604.84,E2 10604.84} C_VEL
LIN {X 0,Y 388.236,Z 654.917,A -85,B 0,C 180,E1 10602.036,E2 10602.036} C_VEL
